fbOEERejectionReason1(
                        bEnable				:= TRUE,
                        bReset				:= ,
                        udiGlobalCounter	:= VIS.udiCounterGlobal, //Globalny licznik konfekcji [szt]
                        bAddReason			:= P13_BottleTransfer.fbBottleTransfer.eRunningState>1 AND VIS.nBottleTransferPlaceOption=2, // może dodać dodatkowy warunek?
                        bReason1			:= eRobotPackageState[1].bWeightTooLow 			AND eRobotPackageState[1].bBottlePresent,
                        sReason1Description	:= 'WZM',
                        bReason2			:= eRobotPackageState[1].bWeightTooHigh 		AND eRobotPackageState[1].bBottlePresent,
                        sReason2Description	:= 'WZD',
                        bReason3			:= NOT eRobotPackageState[1].bCapOK 			AND eRobotPackageState[1].bBottlePresent,
                        sReason3Description	:= 'BNPZ',
                        bReason4			:= NOT eRobotPackageState[1].bCapGripperScrewed AND eRobotPackageState[1].bBottlePresent,
                        sReason4Description	:= 'NZZSZ',
                        bReason5			:= NOT eRobotPackageState[1].bCapCorrectCapOn 	AND eRobotPackageState[1].bBottlePresent,
                        sReason5Description	:= 'BNZZ',
                        bReason6			:= eRobotPackageState[1].bCapCorrectNOK 		AND eRobotPackageState[1].bBottlePresent,
                        sReason6Description	:= 'NZZ',
                        bReason7			:=, 
                        sReason7Description	:= ,      
                        sRejectionReason	:= sOEERejectionReason1Temp,
                        );

fbOEERejectionReason2(
                        bEnable				:= TRUE,
                        bReset				:= ,
                        udiGlobalCounter	:= VIS.udiCounterGlobal, //Globalny licznik konfekcji [szt]
                        bAddReason			:= P13_BottleTransfer.fbBottleTransfer.eRunningState>1 AND VIS.nBottleTransferPlaceOption=2,
                        bReason1			:= eRobotPackageState[2].bWeightTooLow 			AND eRobotPackageState[2].bBottlePresent,
                        sReason1Description	:= 'WZM',
                        bReason2			:= eRobotPackageState[2].bWeightTooHigh 		AND eRobotPackageState[2].bBottlePresent,
                        sReason2Description	:= 'WZD',
                        bReason3			:= NOT eRobotPackageState[2].bCapOK 			AND eRobotPackageState[2].bBottlePresent,
                        sReason3Description	:= 'BNPZ',
                        bReason4			:= NOT eRobotPackageState[2].bCapGripperScrewed AND eRobotPackageState[2].bBottlePresent,
                        sReason4Description	:= 'NZZSZ',
                        bReason5			:= NOT eRobotPackageState[2].bCapCorrectCapOn 	AND eRobotPackageState[2].bBottlePresent,
                        sReason5Description	:= 'BNZZ',
                        bReason6			:= eRobotPackageState[2].bCapCorrectNOK 		AND eRobotPackageState[2].bBottlePresent,
                        sReason6Description	:= 'NZZ',
                        bReason7			:= , 
                        sReason7Description	:= ,      
                        sRejectionReason	:= sOEERejectionReason2Temp,
                        );
						
	rtfbOEERejectionReason2bDone(CLK:=fbOEERejectionReason2.bDone,Q=>);
	rtfbOEERejectionReason1bDone(CLK:=fbOEERejectionReason1.bDone,Q=>);
// dodałem na testy! 20.06	
	IF rtfbOEERejectionReason1bDone.Q AND  VIS.nBottleTransferPickOption=1 THEN
		VIS.sOEERejectionReason 			:=sOEERejectionReason1Temp;//	CONCAT(sOEERejectionReason1Temp,';');
		irtfbOEERejectionReason1bDoneCount	:=	irtfbOEERejectionReason1bDoneCount+1;
	END_IF
	
	
	IF rtfbOEERejectionReason2bDone.Q AND  VIS.nBottleTransferPickOption=2 THEN
		VIS.sOEERejectionReason 			:=	CONCAT(CONCAT(sOEERejectionReason1Temp,';'),sOEERejectionReason2Temp);
		irtfbOEERejectionReason2bDoneCount	:=	irtfbOEERejectionReason2bDoneCount+1;
	END_IF
	
    //Przeniesione dodawanie liczników, po to żeby dla wizualizacji i skryptów było łatwiej (kolejnosć odczytu)
    IF bAddGlobalCounter AND (fbOEERejectionReason2.bDone OR fbOEERejectionReason1.bDone )THEN
        VIS.uiCounterBadBottles                	:= VIS.uiCounterBadBottles		+ INT_TO_UINT(P00_PackML.nCounterFormsToLoad);//+ 1;// czy aby na pewno +1 ???
        VIS.udiCounterGlobalBadBottles        	:= VIS.udiCounterGlobalBadBottles	+ INT_TO_UDINT(P00_PackML.nCounterFormsToLoad);
        VIS.udiCounterGlobal                   	:= VIS.udiCounterGlobal			+ INT_TO_UDINT(P00_PackML.nCounterFormsToLoad);
        //VIS.udiCounterShiftBottles            	:= VIS.udiCounterShiftBottles	+ INT_TO_UDINT(P00_PackML.nCounterFormsToLoad);
        bAddGlobalCounter                    	:= FALSE;
    END_IF

    IF fbOEERejectionReason1.bAddReason THEN
       ifbOEERejectionReason1bAddReasonCount:=ifbOEERejectionReason1bAddReasonCount+1;
    END_IF
	
    IF fbOEERejectionReason2.bAddReason THEN
        ifbOEERejectionReason2bAddReasonCount:=ifbOEERejectionReason2bAddReasonCount+1;
     END_IF
END_ACTION

END_PROGRAM

// ---- POUs/FB/FB_OEECycleTimes.TcPOU
(*
Nazwa:			FB_OEECycleTimes
Opis:			czasy cyklów
Wersja:			v0.1
Data:			2021-11-09
Autor:			DP
Urzadzenia:		
Konfiguracja:	
Info: 
- dodano opcje przesuwu liniowego
*)
FUNCTION_BLOCK FB_OEECycleTimes
VAR_INPUT
	bEnable: BOOL;				//Zezwolenie na pracę
	bReset:BOOL;				//Stop awaryjny nieaktywny
	tStation1CT:TIME;			//Czas cyklu stacji nr 1
	bStation1En:BOOL;			//Zezwolenie pracy stacji nr 1
	sStation1Name:STRING;		//Nazwa stacji nr 1
	tStation2CT:TIME;			//Czas cyklu stacji nr 2
	bStation2En:BOOL;			//Zezwolenie pracy stacji nr 2
	sStation2Name:STRING;		//Nazwa stacji nr 2
	tStation3CT:TIME;			//Czas cyklu stacji nr 3
	bStation3En:BOOL;			//Zezwolenie pracy stacji nr 3
	sStation3Name:STRING;		//Nazwa stacji nr 3
	tStation4CT:TIME;			//Czas cyklu stacji nr 4
	bStation4En:BOOL;			//Zezwolenie pracy stacji nr 4
	sStation4Name:STRING;		//Nazwa stacji nr 4
	tStation5CT:TIME;			//Czas cyklu stacji nr 5
	bStation5En:BOOL;			//Zezwolenie pracy stacji nr 5
	sStation5Name:STRING;		//Nazwa stacji nr 5
	tStation6CT:TIME;			//Czas cyklu stacji nr 6
	bStation6En:BOOL;			//Zezwolenie pracy stacji nr 6
	sStation6Name:STRING;		//Nazwa stacji nr 6
	tStation7CT:TIME;			//Czas cyklu stacji nr 7
	bStation7En:BOOL;			//Zezwolenie pracy stacji nr 7
	sStation7Name:STRING;		//Nazwa stacji nr 7
	tStation8CT:TIME;			//Czas cyklu stacji nr 8
	bStation8En:BOOL;			//Zezwolenie pracy stacji nr 8
	sStation8Name:STRING;		//Nazwa stacji nr 8
	tStation9CT:TIME;			//Czas cyklu stacji nr 9
	bStation9En:BOOL;			//Zezwolenie pracy stacji nr 9
	sStation9Name:STRING;		//Nazwa stacji nr 9
	tStation10CT:TIME;			//Czas cyklu stacji nr 10
	bStation10En:BOOL;			//Zezwolenie pracy stacji nr 10
	sStation10Name:STRING;		//Nazwa stacji nr 10
	tStation11CT:TIME;			//Czas cyklu stacji nr 11
	bStation11En:BOOL;			//Zezwolenie pracy stacji nr 11
	sStation11Name:STRING;		//Nazwa stacji nr 11
	tStation12CT:TIME;			//Czas cyklu stacji nr 12
	bStation12En:BOOL;			//Zezwolenie pracy stacji nr 12
	sStation12Name:STRING;		//Nazwa stacji nr 12
	tStation13CT:TIME;			//Czas cyklu stacji nr 13
	bStation13En:BOOL;			//Zezwolenie pracy stacji nr 13
	sStation13Name:STRING;		//Nazwa stacji nr 13
	tStation14CT:TIME;			//Czas cyklu stacji nr 14
	bStation14En:BOOL;			//Zezwolenie pracy stacji nr 14
	sStation14Name:STRING;		//Nazwa stacji nr 14
	tStation15CT:TIME;			//Czas cyklu stacji nr 15
	bStation15En:BOOL;			//Zezwolenie pracy stacji nr 15	
	sStation15Name:STRING;		//Nazwa stacji nr 15
	tStation16CT:TIME;			//Czas cyklu stacji nr 16
	bStation16En:BOOL;			//Zezwolenie pracy stacji nr 16	
	sStation16Name:STRING;		//Nazwa stacji nr 16
	tStation17CT:TIME;			//Czas cyklu stacji nr 17
	bStation17En:BOOL;			//Zezwolenie pracy stacji nr 17	
	sStation17Name:STRING;		//Nazwa stacji nr 17
	tStation18CT:TIME;			//Czas cyklu stacji nr 18
	bStation18En:BOOL;			//Zezwolenie pracy stacji nr 18	
	sStation18Name:STRING;		//Nazwa stacji nr 18
	tStation19CT:TIME;			//Czas cyklu stacji nr 19
	bStation19En:BOOL;			//Zezwolenie pracy stacji nr 19	
	sStation19Name:STRING;		//Nazwa stacji nr 19
	tStation20CT:TIME;			//Czas cyklu stacji nr 20
	bStation20En:BOOL;			//Zezwolenie pracy stacji nr 20	
	sStation20Name:STRING;		//Nazwa stacji nr 20
	tStation21CT:TIME;			//Czas cyklu stacji nr 21
	bStation21En:BOOL;			//Zezwolenie pracy stacji nr 21	
	sStation21Name:STRING;		//Nazwa stacji nr 21	
	tStation22CT:TIME;			//Czas cyklu stacji nr 22
	bStation22En:BOOL;			//Zezwolenie pracy stacji nr 22	
	sStation22Name:STRING;		//Nazwa stacji nr 22	
	tStation23CT:TIME;			//Czas cyklu stacji nr 23
	bStation23En:BOOL;			//Zezwolenie pracy stacji nr 23	
	sStation23Name:STRING;		//Nazwa stacji nr 23	
	tStation24CT:TIME;			//Czas cyklu stacji nr 24
	bStation24En:BOOL;			//Zezwolenie pracy stacji nr 24	
	sStation24Name:STRING;		//Nazwa stacji nr 24	
	tStation25CT:TIME;			//Czas cyklu stacji nr 25
	bStation25En:BOOL;			//Zezwolenie pracy stacji nr 25	
	sStation25Name:STRING;		//Nazwa stacji nr 25	
	tStation26CT:TIME;			//Czas cyklu stacji nr 26
	bStation26En:BOOL;			//Zezwolenie pracy stacji nr 26	
	sStation26Name:STRING;		//Nazwa stacji nr 26	
	tStation27CT:TIME;			//Czas cyklu stacji nr 27
	bStation27En:BOOL;			//Zezwolenie pracy stacji nr 27	
	sStation27Name:STRING;		//Nazwa stacji nr 27	
	tStation28CT:TIME;			//Czas cyklu stacji nr 28
	bStation28En:BOOL;			//Zezwolenie pracy stacji nr 28	
	sStation28Name:STRING;		//Nazwa stacji nr 28	
	tStation29CT:TIME;			//Czas cyklu stacji nr 29
	bStation29En:BOOL;			//Zezwolenie pracy stacji nr 29	
	sStation29Name:STRING;		//Nazwa stacji nr 29	
	tStation30CT:TIME;			//Czas cyklu stacji nr 30
	bStation30En:BOOL;			//Zezwolenie pracy stacji nr 30	
	sStation30Name:STRING;		//Nazwa stacji nr 30	
	tStation31CT:TIME;			//Czas cyklu stacji nr 31
	bStation31En:BOOL;			//Zezwolenie pracy stacji nr 31	
	sStation31Name:STRING;		//Nazwa stacji nr 31	
	
END_VAR
VAR_OUTPUT
	AsCycleTimes					:ARRAY [0..63] OF STRING;		// Tabela czasów cykli 		[symbol_stacji;czas_w_ms]
END_VAR

VAR

END_VAR

ErrorHandling();
Cycle();
ManualMovements();
Statistics();

ACTION Cycle:


//Generowanie tablicy
IF tStation1CT < T#10S THEN	AsCycleTimes[1]:=	CONCAT(sStation1Name,	CONCAT(';',DINT_TO_STRING(TIME_TO_DINT(tStation1CT))));		ELSE tStation1CT := T#10S; END_IF;

IF tStation2CT < T#10S THEN	AsCycleTimes[2]:=	CONCAT(sStation2Name,	CONCAT(';',DINT_TO_STRING(TIME_TO_DINT(tStation2CT))));		ELSE tStation1CT := T#10S; END_IF;

IF tStation3CT < T#10S THEN	AsCycleTimes[3]:=	CONCAT(sStation3Name,	CONCAT(';',DINT_TO_STRING(TIME_TO_DINT(tStation3CT))));		ELSE tStation1CT := T#10S; END_IF;

IF tStation4CT < T#10S THEN	AsCycleTimes[4]:=	CONCAT(sStation4Name,	CONCAT(';',DINT_TO_STRING(TIME_TO_DINT(tStation4CT))));		ELSE tStation4CT := T#10S; END_IF;

IF tStation5CT < T#10S THEN	AsCycleTimes[5]:=	CONCAT(sStation5Name,	CONCAT(';',DINT_TO_STRING(TIME_TO_DINT(tStation5CT))));		ELSE tStation5CT := T#10S; END_IF;

IF tStation6CT < T#10S THEN	AsCycleTimes[6]:=	CONCAT(sStation6Name,	CONCAT(';',DINT_TO_STRING(TIME_TO_DINT(tStation6CT))));		ELSE tStation6CT := T#10S; END_IF;
	
IF tStation7CT < T#10S THEN AsCycleTimes[7]:=	CONCAT(sStation7Name,	CONCAT(';',DINT_TO_STRING(TIME_TO_DINT(tStation7CT))));		ELSE tStation7CT := T#10S; END_IF;
	
IF tStation8CT < T#10S THEN AsCycleTimes[8]:=	CONCAT(sStation8Name,	CONCAT(';',DINT_TO_STRING(TIME_TO_DINT(tStation8CT))));		ELSE tStation8CT := T#10S; END_IF;
	
IF tStation9CT < T#10S THEN AsCycleTimes[9]:=	CONCAT(sStation9Name,	CONCAT(';',DINT_TO_STRING(TIME_TO_DINT(tStation9CT))));		ELSE tStation9CT := T#10S; END_IF;
	
IF tStation10CT < T#10S THEN AsCycleTimes[10]:=	CONCAT(sStation10Name,	CONCAT(';',DINT_TO_STRING(TIME_TO_DINT(tStation10CT))));	ELSE tStation10CT := T#10S; END_IF;

IF tStation11CT < T#10S THEN AsCycleTimes[11]:=	CONCAT(sStation11Name,	CONCAT(';',DINT_TO_STRING(TIME_TO_DINT(tStation11CT))));	ELSE tStation11CT := T#10S; END_IF;

IF tStation12CT < T#10S THEN AsCycleTimes[12]:=	CONCAT(sStation12Name,	CONCAT(';',DINT_TO_STRING(TIME_TO_DINT(tStation12CT))));	ELSE tStation12CT := T#10S; END_IF;

IF tStation13CT < T#10S THEN AsCycleTimes[13]:=	CONCAT(sStation13Name,	CONCAT(';',DINT_TO_STRING(TIME_TO_DINT(tStation13CT))));	ELSE tStation13CT := T#10S; END_IF;

IF tStation14CT < T#10S THEN AsCycleTimes[14]:=	CONCAT(sStation14Name,	CONCAT(';',DINT_TO_STRING(TIME_TO_DINT(tStation14CT))));	ELSE tStation14CT := T#10S; END_IF;

IF tStation15CT < T#10S THEN AsCycleTimes[15]:=	CONCAT(sStation15Name,	CONCAT(';',DINT_TO_STRING(TIME_TO_DINT(tStation15CT))));	ELSE tStation15CT := T#10S; END_IF;

IF tStation16CT < T#10S THEN AsCycleTimes[16]:=	CONCAT(sStation16Name,	CONCAT(';',DINT_TO_STRING(TIME_TO_DINT(tStation16CT))));	ELSE tStation16CT := T#10S; END_IF;

IF tStation17CT < T#10S THEN AsCycleTimes[17]:=	CONCAT(sStation17Name,	CONCAT(';',DINT_TO_STRING(TIME_TO_DINT(tStation17CT))));	ELSE tStation17CT := T#10S; END_IF;

IF tStation18CT < T#10S THEN AsCycleTimes[18]:=	CONCAT(sStation18Name,	CONCAT(';',DINT_TO_STRING(TIME_TO_DINT(tStation18CT))));	ELSE tStation18CT := T#10S; END_IF;

IF tStation19CT < T#10S THEN AsCycleTimes[19]:=	CONCAT(sStation19Name,	CONCAT(';',DINT_TO_STRING(TIME_TO_DINT(tStation19CT))));	ELSE tStation19CT := T#10S; END_IF;

IF tStation20CT < T#10S THEN AsCycleTimes[20]:=	CONCAT(sStation20Name,	CONCAT(';',DINT_TO_STRING(TIME_TO_DINT(tStation20CT))));	ELSE tStation20CT := T#10S; END_IF;

IF tStation21CT < T#10S THEN AsCycleTimes[21]:=	CONCAT(sStation21Name,	CONCAT(';',DINT_TO_STRING(TIME_TO_DINT(tStation21CT))));	ELSE tStation21CT := T#10S; END_IF;

IF tStation22CT < T#10S THEN AsCycleTimes[22]:=	CONCAT(sStation22Name,	CONCAT(';',DINT_TO_STRING(TIME_TO_DINT(tStation22CT))));	ELSE tStation22CT := T#10S; END_IF;

IF tStation23CT < T#10S THEN AsCycleTimes[23]:=	CONCAT(sStation23Name,	CONCAT(';',DINT_TO_STRING(TIME_TO_DINT(tStation23CT))));	ELSE tStation23CT := T#10S; END_IF;
	
IF tStation24CT < T#10S THEN AsCycleTimes[24]:=	CONCAT(sStation24Name,	CONCAT(';',DINT_TO_STRING(TIME_TO_DINT(tStation24CT))));	ELSE tStation24CT := T#10S; END_IF;

IF tStation25CT < T#10S THEN AsCycleTimes[25]:=	CONCAT(sStation25Name,	CONCAT(';',DINT_TO_STRING(TIME_TO_DINT(tStation25CT))));	ELSE tStation25CT := T#10S; END_IF;

IF tStation26CT < T#10S THEN AsCycleTimes[26]:=	CONCAT(sStation26Name,	CONCAT(';',DINT_TO_STRING(TIME_TO_DINT(tStation26CT))));	ELSE tStation26CT := T#10S; END_IF;

IF tStation27CT < T#10S THEN AsCycleTimes[27]:=	CONCAT(sStation27Name,	CONCAT(';',DINT_TO_STRING(TIME_TO_DINT(tStation27CT))));	ELSE tStation27CT := T#10S; END_IF;

IF tStation28CT < T#10S THEN AsCycleTimes[28]:=	CONCAT(sStation28Name,	CONCAT(';',DINT_TO_STRING(TIME_TO_DINT(tStation28CT))));	ELSE tStation28CT := T#10S; END_IF;

IF tStation29CT < T#10S THEN AsCycleTimes[29]:=	CONCAT(sStation29Name,	CONCAT(';',DINT_TO_STRING(TIME_TO_DINT(tStation29CT))));	ELSE tStation29CT := T#10S; END_IF;

IF tStation30CT < T#10S THEN AsCycleTimes[30]:=	CONCAT(sStation30Name,	CONCAT(';',DINT_TO_STRING(TIME_TO_DINT(tStation30CT))));	ELSE tStation30CT := T#10S; END_IF;

IF tStation31CT < T#10S THEN AsCycleTimes[31]:=	CONCAT(sStation31Name,	CONCAT(';',DINT_TO_STRING(TIME_TO_DINT(tStation31CT))));	ELSE tStation31CT := T#10S; END_IF;
END_ACTION

ACTION ErrorHandling:

END_ACTION

ACTION ManualMovements:

END_ACTION

ACTION Statistics:

END_ACTION

END_FUNCTION_BLOCK

// ---- POUs/FB/FB_OEERejectionReason.TcPOU
(*
Nazwa:			FB_OEERejectionReasons
Opis:			Powód odrzuceń 
Wersja:			v0.1
Data:			2019-12-17
Autor:			DP
Urzadzenia:		
Konfiguracja:	
Info: 
- 
*)
FUNCTION_BLOCK FB_OEERejectionReason
VAR_INPUT
	bEnable: BOOL;				//Zezwolenie na pracę
	bReset:BOOL;				//Stop awaryjny nieaktywny
	udiGlobalCounter:UDINT;		//Globalny licznik
	bAddReason:BOOL;			//Dodaj pomiar
	bReason1:BOOL;
	sReason1Description:STRING;	//Nazwa stacji nr 1
	bReason2:BOOL;
	sReason2Description:STRING;	//Nazwa stacji nr 2
	bReason3:BOOL;
	sReason3Description:STRING;	//Nazwa stacji nr 3
	bReason4:BOOL;
	sReason4Description:STRING;	//Nazwa stacji nr 4
	bReason5:BOOL;
	sReason5Description:STRING;	//Nazwa stacji nr 5
	bReason6:BOOL;
	sReason6Description:STRING;	//Nazwa stacji nr 6
	bReason7:BOOL;
	sReason7Description:STRING;	//Nazwa stacji nr 7
	bReason8:BOOL;
	sReason8Description:STRING;	//Nazwa stacji nr 8
	bReason9:BOOL;
	sReason9Description:STRING;	//Nazwa stacji nr 9
	bReason10:BOOL;
	sReason10Description:STRING;	//Nazwa stacji nr 10
	bReason11:BOOL;
	sReason11Description:STRING;	//Nazwa stacji nr 11
	bReason12:BOOL;
	sReason12Description:STRING;	//Nazwa stacji nr 12
	bReason13:BOOL;
	sReason13Description:STRING;	//Nazwa stacji nr 13
	bReason14:BOOL;
	sReason14Description:STRING;	//Nazwa stacji nr 14
END_VAR

VAR_IN_OUT
	sRejectionReason			:STRING;		// Powodu odrzuceń	[symbol_odrzucenia] narazie tylko w tabeli 1
END_VAR
VAR_OUTPUT
	bDone						:BOOL;		// Powodu odrzuceń	[symbol_odrzucenia] narazie tylko w tabeli 1
END_VAR

VAR
	rtAddReason: R_TRIG;
	tonResetDone: TON;
END_VAR

ErrorHandling();
Cycle();
ManualMovements();
Statistics();

ACTION Cycle:
tonResetDone(IN:=bDone,PT:=T#300MS);
rtAddReason(CLK:=bAddReason,Q=>);
IF rtAddReason.Q THEN
	IF bReason1 THEN
		sRejectionReason:= sReason1Description;
	ELSIF bReason2 THEN		                
		sRejectionReason:= sReason2Description;
	ELSIF bReason3 THEN		                
		sRejectionReason:= sReason3Description;
	ELSIF bReason4 THEN		                
		sRejectionReason:= sReason4Description;
	ELSIF bReason5 THEN		                
		sRejectionReason:= sReason5Description;
	ELSIF bReason6 THEN		                
		sRejectionReason:= sReason6Description;
	ELSIF bReason7 THEN		                
		sRejectionReason:= sReason7Description;
	ELSIF bReason8 THEN		                
		sRejectionReason:= sReason8Description;
	ELSIF bReason9 THEN		                
		sRejectionReason:= sReason9Description;
	ELSIF bReason10 THEN		                
		sRejectionReason:= sReason10Description;
	ELSIF bReason11 THEN		                
		sRejectionReason:= sReason11Description;
	ELSIF bReason12 THEN		                
		sRejectionReason:= sReason12Description;
	ELSIF bReason13 THEN		                
		sRejectionReason:= sReason13Description;
	ELSIF bReason14 THEN		                
		sRejectionReason:= sReason14Description;

	END_IF
	bDone:= TRUE;
END_IF
IF tonResetDone.Q THEN
	bDone:= FALSE;
END_IF
END_ACTION

ACTION ErrorHandling:

END_ACTION

ACTION ManualMovements:

END_ACTION

ACTION Statistics:

END_ACTION

END_FUNCTION_BLOCK

// ---- POUs/P00_Recipes.TcPOU
PROGRAM P00_Recipes
(*
Nazwa:			P_Recipes
Wersja:			v0.1 			
Autor:			TW,DP
Urzadzenia:		HMI, 
Konfiguracja:	
Info:
- 50 receptur
- sortowanie
- odczytwanie, zapisywanie jako nowa, aktualizacja, usuwanie, wybór
- receptura 1 jako ustawienia fabryczne
Uwagi:
- na końcu aktualizować nastawy pierwszej receptury
Zmiany:
2018-05-07 DP Dodano na stałe wpisywanie danych do pierwszej receptury
*)
VAR
	i: INT;
	h: INT;
	bTestDwuFaz: BOOL;
	iLidSealerTempHisteresis: INT;
	bTestTransporter: BOOL;
	fbiPackageNozzleDiameter:FB_Skalowanie;
	rPackageNozzleDiameterFactor:REAL;	
	rPackageMassTypeFactor:REAL;	
END_VAR

//wybór programu
IF VIS.bChooseRecipe THEN
	IF VIS.bDialogBoxAck THEN
		VIS.bChooseRecipe := FALSE;
		VIS.bDialogBoxAck:=FALSE;
		bRecipeAfterPowerStateChosen := TRUE; //Wybrano pierwszą recepturę po ruchomieniu
	ELSIF VIS.bDialogBoxCancelAck THEN
		VIS.bDialogBoxAck:=FALSE;
		VIS.bChooseRecipe := FALSE;
		VIS.bDialogBoxCancelAck:=FALSE;
	END_IF
END_IF

(*Automatyczne ustawianie danych receptur*)
aAutoSetRecipeParameters();

(*dane receptur*)
aShowToAll();
aTwoSpeeds();
aLimits();	
//Receptura fabryczna
//Na stałe bez możliwości zmiany
//Zawsze można zapisać jako inną i tam zmieniać parametry
VIS.bChooseRecipe;
VIS.bDialogBoxAck;
IF NOT bFirstPositioningDone  THEN						//do skomentowania Vasyl
	aFactoryRecipes();
END_IF
IF bHomingCanceled AND NOT bFirstPositioningDone THEN
	bFirstPositioningDone	:= TRUE;
END_IF

ACTION aAutoSetRecipeParameters:

(****************** AUTO DOSTRAJANIE CZASÓW TRANSPORTERÓW*********)
	//Czas przy najwolnejszej prędkości transportera 15Hz
	//15Hz 300 2000ms
	//25Hz 500 1300ms
	//35Hz 700 1000ms
	//45Hz 900 700ms
	//56Hz 1100 600ms
	//67Hz 1300 500ms
	// Wyznaczona funkcja potęgowa
	IF GVL.nFormTransportersDispencerVelocitySV > 0 AND GVL.nFormTransportersDispencerVelocitySV <1000 THEN
		
		VIS.nGateBeforeDispencersTimeFormInsertingShow := 500;
		(*nExitWheelFormsTime := LREAL_TO_UINT(
										850601 * EXPT(nFormTransportersVelocitySV,-0.94)
											);*)										
		{warning 'Czasy otwarcia narazie na stałe-sprawdzić dla szybkiej i najwolniejszej prędkości transportera}			
	ELSE
		VIS.nGateBeforeDispencersTimeFormInsertingShow := 300;
		(*nExitWheelFormsTime := LREAL_TO_UINT(
										850601 * EXPT(nFormTransportersVelocitySV,-0.94)
											);*)										
			;
	END_IF
	
	IF 		GVL.nFormTransportersDispencerVelocitySV 	>	1100	THEN			
				VIS.nGateRobotTimeFormInsertingShow		:= 300;	//bylo 300	
	ELSIF 		GVL.nFormTransportersDispencerVelocitySV 	>	1000	THEN			
				VIS.nGateRobotTimeFormInsertingShow		:= 300;		
	ELSIF	GVL.nFormTransportersDispencerVelocitySV 	>	900		THEN
				VIS.nGateRobotTimeFormInsertingShow		:= 400;		
	ELSIF	GVL.nFormTransportersDispencerVelocitySV 	>	800		THEN
				VIS.nGateRobotTimeFormInsertingShow		:= 450;		
	ELSIF	GVL.nFormTransportersDispencerVelocitySV 	>	700		THEN
				VIS.nGateRobotTimeFormInsertingShow		:= 600;	
	ELSIF	GVL.nFormTransportersDispencerVelocitySV 	>	600		THEN
				VIS.nGateRobotTimeFormInsertingShow		:= 800;	
	ELSIF	GVL.nFormTransportersDispencerVelocitySV 	>	500		THEN
				VIS.nGateRobotTimeFormInsertingShow		:= 900;	
	ELSE
			VIS.nGateRobotTimeFormInsertingShow		:= 1000;	
	END_IF	
	
	
	
	//Parametry opakowania  [Ekran obliczania parametrów]
    //[[[[[[[[[[[[[[[[[[[[[[[[[[[[[[[[[[[[[[[[[[[[[[[[[[[
 	VIS.iPackagePuckInsertHeightShow;// Wysokość wkładki w formatce (0-100mm)  (samej wkładki) (Do pozycji odkładania robota)              
  	VIS.iPackageMassTypeShow		;// Typ masy 	(0-Woda, 1-Olej, 2-Mydło, 3-Krem itd.)
	VIS.iPackageCapTypeShow			;// Typ nasadki (0-Fliptop, 1-Pompka/Atomizer, 2-Kulka, 3-Airless, 4-, 5- Deko, 6-Nakrętka_słoika
	VIS.iPackageCapDiameterShow		;// Średnica nasadki (5-100mm),
	VIS.iPackageHeightShow			;// Wysokość butelki razem z formatką (50-300mm),	
	VIS.iPackageCappedHeightShow	;// Wysokość butelki razem z dokręconą nakrętką i formatką (50-350mm),		
	VIS.iPackageNozzleDiameterShow	;// Srednica zewnetrzna wylewki (5-30mm),	
	VIS.lrDispencer1DoseVolumeShow  ;// Ilość dozy (10-560ml)
 	VIS.lrCupWeightShow	 			;// Waga opakowania (0-500g)
 	VIS.bRecipeCalculate;			 // Oblicz
	 //[[[[[[[[[[[[[[[[[[[[[[[[[[[[[[[[[[[[[[[[[[[[[[[[[[[
	 
	// Limity
	 IF VIS.iPackageHeightShow = 0 			THEN VIS.iPackageHeightShow := 150;	 			END_IF
	 IF VIS.iPackageCappedHeightShow = 0 	THEN VIS.iPackageCappedHeightShow := 160;		END_IF	 
	 IF VIS.iPackageNozzleDiameterShow = 0 	THEN VIS.iPackageNozzleDiameterShow := 16;		END_IF	 
	
	// Skalowanie - Prędkość Dozowania <-> Średnica wylewki
	 rPackageNozzleDiameterFactor := 						1.4285 * EXPT(VIS.iPackageNozzleDiameterShow,1.5615);	
	// Skalowanie - Typ masy 	(0-Woda, 1-Olej, 2-Mydło, 3-Krem itd.)
	IF   	VIS.iPackageMassTypeShow	= 0 THEN	rPackageMassTypeFactor := 1.0;
	ELSIF	VIS.iPackageMassTypeShow	= 1 THEN	rPackageMassTypeFactor := 0.8;
	ELSIF	VIS.iPackageMassTypeShow	= 2 THEN	rPackageMassTypeFactor := 1.3;
	ELSIF	VIS.iPackageMassTypeShow	= 3 THEN	rPackageMassTypeFactor := 1.5;		END_IF
	// Prędkość dozowania
	rPackageNozzleDiameterFactor; (**) rPackageMassTypeFactor;
	
	// Oblicz
	IF VIS.bRecipeCalculate THEN
					
        //Podawanie butelekButelki                                  
		VIS.lrPucksInserterHammerHeightSVShow				:=	VIS.iPackageHeightShow+1;                                            				                                                                                                                           																		
       
		//Dozownik	                             	                                                                                     												
		VIS.lrDispencersLifterReadyPositionShow				:=	VIS.iPackageHeightShow + 60;                                                                                             
		VIS.lrDispencer1LifterStartDosePositionShow			:=	VIS.iPackagePuckInsertHeightShow + 29 + 25;                                           
		VIS.lrDispencer1LifterStopDosePositionShow			:=	VIS.iPackageHeightShow - 10;                                                                                  
		VIS.lrDispencersCatchHeightSVShow					:=	VIS.iPackageHeightShow - 5;                                                  
       	IF  VIS.iPackageMassTypeShow = 0 THEN // (0-Woda, 1-Olej, 2-Mydło, 3-Krem itd.)                               
			VIS.lrDispencer1Phase1VolumeShow				:=	FLOOR(VIS.lrDispencer1DoseVolumeShow*0.2);                                          
			VIS.lrDispencer1Phase2VolumeShow				:=	0;
			VIS.lrDispencer1Phase1VelocityShow				:=	rPackageNozzleDiameterFactor * rPackageMassTypeFactor * 0.7;
			VIS.lrDispencer1Phase2VelocityShow				:=	rPackageNozzleDiameterFactor * rPackageMassTypeFactor;
			VIS.lrDispencer1Phase3VelocityShow				:=	rPackageNozzleDiameterFactor * rPackageMassTypeFactor * 0.7;
			VIS.lrDispencer1SuckVelocityShow				:=	200;
			VIS.lrDispencer1Phase1AccelerationShow			:=	300;
			VIS.lrDispencer1Phase2AccelerationShow			:=	400;
			VIS.lrDispencer1Phase3AccelerationShow			:=	50;
			VIS.lrDispencer1SuckAccelerationShow			:=	3000;
			VIS.lrDispencer1Phase1DecelerationShow			:=	150;
			VIS.lrDispencer1Phase2DecelerationShow			:=	1000;
			VIS.lrDispencer1Phase3DecelerationShow			:=	50;
			VIS.udiDispencer1DosingDoneDelayTimeShow		:=	100;
			VIS.lrDispencer1SuckValveOpenVolumeShow			:=	0;
			VIS.lrDispencer1SuckValveOpenTimeDelayShow		:=	0;
			VIS.lrDispencer1SuckValveCloseVolumeShow		:=	0;
			VIS.lrDispencer1SuckValveCloseTimeDelayShow		:=	0;
			VIS.lrDispencer1DoseValveOpenVolumeShow			:=	0;
			VIS.lrDispencer1DoseValveOpenTimeAccShow		:=	100;
			VIS.lrDispencer1DoseValveCloseVolumeShow		:=	0;
			VIS.lrDispencer1DoseValveCloseTimeDecShow		:=	0;
			VIS.lrDispencer1DoseSuckingVolumeShow			:=	0;
			VIS.lrDispencer1DoseSuckingTimeDelayShow		:=	0;
			VIS.bDispencer1DoseSuckingShow					:=	FALSE;
			VIS.bDispencer2LiftSynchroPh1Show				:=	FALSE;
			VIS.bDispencer2LiftSynchroPh2Show				:=	TRUE;
			VIS.bDispencer2LiftSynchroPh3Show				:=	TRUE;	
		ELSIF VIS.iPackageMassTypeShow = 1 THEN // (0-Woda, 1-Olej, 2-Mydło, 3-Krem itd.)   
			VIS.lrDispencer1Phase1VolumeShow				:=	FLOOR(VIS.lrDispencer1DoseVolumeShow*0.2);                                          
			VIS.lrDispencer1Phase2VolumeShow				:=	FLOOR(VIS.lrDispencer1DoseVolumeShow*0.2); 
			VIS.lrDispencer1Phase1VelocityShow				:=	rPackageNozzleDiameterFactor * rPackageMassTypeFactor * 0.7;
			VIS.lrDispencer1Phase2VelocityShow				:=	rPackageNozzleDiameterFactor * rPackageMassTypeFactor;
			VIS.lrDispencer1Phase3VelocityShow				:=	rPackageNozzleDiameterFactor * rPackageMassTypeFactor * 0.7;
			VIS.lrDispencer1SuckVelocityShow				:=	100;
			VIS.lrDispencer1Phase1AccelerationShow			:=	40;
			VIS.lrDispencer1Phase2AccelerationShow			:=	50;
			VIS.lrDispencer1Phase3AccelerationShow			:=	40;
			VIS.lrDispencer1SuckAccelerationShow			:=	500;
			VIS.lrDispencer1Phase1DecelerationShow			:=	80;
			VIS.lrDispencer1Phase2DecelerationShow			:=	100;
			VIS.lrDispencer1Phase3DecelerationShow			:=	80;
			VIS.udiDispencer1DosingDoneDelayTimeShow		:=	200;
			VIS.lrDispencer1SuckValveOpenVolumeShow			:=	0;
			VIS.lrDispencer1SuckValveOpenTimeDelayShow		:=	0;
			VIS.lrDispencer1SuckValveCloseVolumeShow		:=	0;
			VIS.lrDispencer1SuckValveCloseTimeDelayShow		:=	0;
			VIS.lrDispencer1DoseValveOpenVolumeShow			:=	0;
			VIS.lrDispencer1DoseValveOpenTimeAccShow		:=	200;
			VIS.lrDispencer1DoseValveCloseVolumeShow		:=	0;
			VIS.lrDispencer1DoseValveCloseTimeDecShow		:=	0;
			VIS.lrDispencer1DoseSuckingVolumeShow			:=	0;
			VIS.lrDispencer1DoseSuckingTimeDelayShow		:=	0;
			VIS.bDispencer1DoseSuckingShow					:=	FALSE;
			VIS.bDispencer2LiftSynchroPh1Show				:=	TRUE;
			VIS.bDispencer2LiftSynchroPh2Show				:=	TRUE;
			VIS.bDispencer2LiftSynchroPh3Show				:=	TRUE;	
		ELSIF VIS.iPackageMassTypeShow = 2 THEN // (0-Woda, 1-Olej, 2-Mydło, 3-Krem itd.)   
			VIS.lrDispencer1Phase1VolumeShow				:=	FLOOR(VIS.lrDispencer1DoseVolumeShow*0.2);                                          
			VIS.lrDispencer1Phase2VolumeShow				:=	0;
			VIS.lrDispencer1Phase1VelocityShow				:=	rPackageNozzleDiameterFactor * rPackageMassTypeFactor * 0.7;
			VIS.lrDispencer1Phase2VelocityShow				:=	rPackageNozzleDiameterFactor * rPackageMassTypeFactor;      
			VIS.lrDispencer1Phase3VelocityShow				:=	rPackageNozzleDiameterFactor * rPackageMassTypeFactor * 0.7;
			VIS.lrDispencer1SuckVelocityShow				:=	200;
			VIS.lrDispencer1Phase1AccelerationShow			:=	300;
			VIS.lrDispencer1Phase2AccelerationShow			:=	400;
			VIS.lrDispencer1Phase3AccelerationShow			:=	50;
			VIS.lrDispencer1SuckAccelerationShow			:=	3000;
			VIS.lrDispencer1Phase1DecelerationShow			:=	150;
			VIS.lrDispencer1Phase2DecelerationShow			:=	1000;
			VIS.lrDispencer1Phase3DecelerationShow			:=	50;
			VIS.udiDispencer1DosingDoneDelayTimeShow		:=	200;
			VIS.lrDispencer1SuckValveOpenVolumeShow			:=	0;
			VIS.lrDispencer1SuckValveOpenTimeDelayShow		:=	0;
			VIS.lrDispencer1SuckValveCloseVolumeShow		:=	0;
			VIS.lrDispencer1SuckValveCloseTimeDelayShow		:=	0;
			VIS.lrDispencer1DoseValveOpenVolumeShow			:=	0;
			VIS.lrDispencer1DoseValveOpenTimeAccShow		:=	200;
			VIS.lrDispencer1DoseValveCloseVolumeShow		:=	0;
			VIS.lrDispencer1DoseValveCloseTimeDecShow		:=	0;
			VIS.lrDispencer1DoseSuckingVolumeShow			:=	0;
			VIS.lrDispencer1DoseSuckingTimeDelayShow		:=	0;
			VIS.bDispencer1DoseSuckingShow					:=	FALSE;
			VIS.bDispencer2LiftSynchroPh1Show				:=	FALSE;
			VIS.bDispencer2LiftSynchroPh2Show				:=	TRUE;
			VIS.bDispencer2LiftSynchroPh3Show				:=	TRUE;	
		ELSIF VIS.iPackageMassTypeShow = 3 THEN // (0-Woda, 1-Olej, 2-Mydło, 3-Krem itd.)   
			VIS.lrDispencer1Phase1VolumeShow				:=	FLOOR(VIS.lrDispencer1DoseVolumeShow*0.2);                                          
			VIS.lrDispencer1Phase2VolumeShow				:=	0;
			VIS.lrDispencer1Phase1VelocityShow				:=	rPackageNozzleDiameterFactor * rPackageMassTypeFactor * 0.7;
			VIS.lrDispencer1Phase2VelocityShow				:=	rPackageNozzleDiameterFactor * rPackageMassTypeFactor;      
			VIS.lrDispencer1Phase3VelocityShow				:=	rPackageNozzleDiameterFactor * rPackageMassTypeFactor * 0.7;
			VIS.lrDispencer1SuckVelocityShow				:=	200;
			VIS.lrDispencer1Phase1AccelerationShow			:=	300;
			VIS.lrDispencer1Phase2AccelerationShow			:=	400;
			VIS.lrDispencer1Phase3AccelerationShow			:=	50;
			VIS.lrDispencer1SuckAccelerationShow			:=	3000;
			VIS.lrDispencer1Phase1DecelerationShow			:=	150;
			VIS.lrDispencer1Phase2DecelerationShow			:=	1000;
			VIS.lrDispencer1Phase3DecelerationShow			:=	50;
			VIS.udiDispencer1DosingDoneDelayTimeShow		:=	200;
			VIS.lrDispencer1SuckValveOpenVolumeShow			:=	0;
			VIS.lrDispencer1SuckValveOpenTimeDelayShow		:=	0;
			VIS.lrDispencer1SuckValveCloseVolumeShow		:=	0;
			VIS.lrDispencer1SuckValveCloseTimeDelayShow		:=	0;
			VIS.lrDispencer1DoseValveOpenVolumeShow			:=	0;
			VIS.lrDispencer1DoseValveOpenTimeAccShow		:=	200;
			VIS.lrDispencer1DoseValveCloseVolumeShow		:=	0;
			VIS.lrDispencer1DoseValveCloseTimeDecShow		:=	0;
			VIS.lrDispencer1DoseSuckingVolumeShow			:=	0;
			VIS.lrDispencer1DoseSuckingTimeDelayShow		:=	0;
			VIS.bDispencer1DoseSuckingShow					:=	FALSE;
			VIS.bDispencer2LiftSynchroPh1Show				:=	FALSE;
			VIS.bDispencer2LiftSynchroPh2Show				:=	TRUE;
			VIS.bDispencer2LiftSynchroPh3Show				:=	TRUE;	
		END_IF

		//Chwytak butelek
		VIS.lrDispencersCatch1ClosedValueShow				:= VIS.iPackageCapDiameterShow-1;
		VIS.lrDispencersCatch1OpenValueShow					:= 58;
		VIS.lrDispencersCatch2ClosedValueShow				:= VIS.iPackageCapDiameterShow+2;
		VIS.lrDispencersCatch2OpenValueShow					:= 60.2;
		VIS.lrDispencersCatch3ClosedValueShow				:= VIS.iPackageCapDiameterShow+2;
		VIS.lrDispencersCatch3OpenValueShow					:= 60.1;
		VIS.lrDispencersCatch4ClosedValueShow				:= VIS.iPackageCapDiameterShow-1;
		VIS.lrDispencersCatch4OpenValueShow					:= 55.6;
		VIS.lrDispencersCatchToleranceShow					:= 15;
	
		//Waga
		VIS.lrWeightMassSVShow								:= VIS.lrDispencer1DoseVolumeShow;
		VIS.lrWeightUpperToleranceShow						:= FLOOR(VIS.lrDispencer1DoseVolumeShow * 0.02);	
		VIS.lrWeightLowerToleranceShow						:= FLOOR(VIS.lrDispencer1DoseVolumeShow * 0.03);	
		                                                                                                                                                                       		                                                                                        
		//Podajnik platynek                                                                     	                                
		VIS.lrLidFeederHeightPosSVShow						:=	VIS.iPackageHeightShow + 5;  				                                
						                            	                            
		//Sprawdzanie platynek				
		VIS.lrLidPuttedCheckHeightSVShow					:=	VIS.iPackageHeightShow + 5;  	 			
					
		//Zgrzewanie				
		VIS.lrLidSealerHeightPosSVShow						:=	VIS.iPackageHeightShow + 5;  								
		
		//ROPP-Podajnik                                    		
		VIS_ROPP.lrROPPFeederHeightPosSVShow				:=	VIS.iPackageHeightShow + 5;                                                      
		//ROPP-Zakrecanie                    		
		VIS_ROPP.lrROPPCappingHeightPosSVShow				:=	VIS.iPackageHeightShow + 5;  
		
		//Podajnik nakrętek
		VIS.lrCapFeederHeightPosSVShow						:=	VIS.iPackageHeightShow + 12;  		

		//Test nasadki	// Typ nasadki (0-Fliptop, 1-Pompka/Atomizer, 2-Kulka, 3-Airless, 4-, 5- Deko, 6-Nakrętka_słoika
		IF 		VIS.iPackageCapTypeShow	= 0 THEN 			VIS.lrCapPuttedCheckHeightPosSVShow	:=	VIS.iPackageHeightShow ;  
		ELSIF 	VIS.iPackageCapTypeShow	= 1 THEN 			VIS.lrCapPuttedCheckHeightPosSVShow	:=	VIS.iPackageHeightShow ;  	
		ELSIF 	VIS.iPackageCapTypeShow	= 2 THEN 			VIS.lrCapPuttedCheckHeightPosSVShow	:=	VIS.iPackageHeightShow ;   
		ELSIF 	VIS.iPackageCapTypeShow	= 3 THEN 			VIS.lrCapPuttedCheckHeightPosSVShow	:=	VIS.iPackageHeightShow ;  
		ELSIF 	VIS.iPackageCapTypeShow	= 4 THEN 			VIS.lrCapPuttedCheckHeightPosSVShow	:=	VIS.iPackageHeightShow ;  
		ELSIF 	VIS.iPackageCapTypeShow	= 5 THEN 			VIS.lrCapPuttedCheckHeightPosSVShow	:=	VIS.iPackageHeightShow ;  
		ELSIF 	VIS.iPackageCapTypeShow	= 6 THEN 			VIS.lrCapPuttedCheckHeightPosSVShow	:=	VIS.iPackageHeightShow ;  
		END_IF	

		//Zakręcarka
		IF 	VIS.iPackageCapTypeShow	= 0 THEN // Typ nasadki (0-Fliptop, 1-Pompka/Atomizer, 2-Kulka, 3-Airless, 4-, 5- Deko, 6-Nakrętka_słoika
			VIS.lrGripperScrewingTightTorqueShow				:=	0.5;
			VIS.lrGripperScrewing2TightTorqueShow				:=	0.5;
			VIS.iGripperScrewer1ToolShow						:=	0; //0-Dwu,1-Trój,2-Kształtowa/DoKulek,3-Wbijająca,4-Zasysająca
			VIS.lrGripperScrewer1VelocityShow					:=	90;
			VIS.nGripperScrewer1TightTimeShow					:=	300;
			VIS.lrGripperScrewerReadyPositionShow				:=	VIS.iPackageHeightShow + 14;	
			VIS.lrGripperScrewerPushingCapPositionShow			:=	VIS.iPackageHeightShow + 14;	
			VIS.lrGripperScrewerScrewingCapPositionShow			:=	VIS.iPackageHeightShow + 14;
			VIS.lrGripperScrewerFindScrewPositionShow			:=	VIS.iPackageHeightShow + 14;	
			VIS.lrGripperScrewerPressureShow					:=	15;
			VIS.lrGripperScrewerCatchPressureShow				:=	7;
			VIS.lrGripperScrewerPressureExhaustLevelShow		:=	100.0;
			VIS.lrGripperScrewerCatchPressureExhaustLevelShow	:=	100.0;
			VIS.lrGripperScrewerTurnoversToFullScrewedShow		:=	1;
			VIS.lrGripperScrewerThreadPitchShow					:=	3;			
			VIS.lrGripperScrewerThreadTimesShow					:=	1.0;		
			VIS.nGripperScrewerCatchHeightSVShow				:=	VIS_M.iPuckHeight + 10;
			VIS.bGripperScrewer1FindScrewShow					:=	FALSE;
			VIS.bGripperScrewer1Option4Show						:=	FALSE;
			VIS.lrGripperScrewer1FindingScrewDegreeShow			:=	260;
			VIS.bGripperScrewer1Option1Show						:=	FALSE;
			VIS.bGripperScrewer1Option2Show						:=	FALSE;
			VIS.bGripperScrewer1Option3Show						:=	TRUE;
			VIS.bGripperScrewer1Option5Show						:=	FALSE;
			VIS.bGripperScrewer1Option6Show						:=	TRUE;
			VIS.bGripperScrewer1Option7Show						:=	TRUE;
		ELSIF VIS.iPackageCapTypeShow	= 1 THEN // Typ nasadki (0-Fliptop, 1-Pompka/Atomizer, 2-Kulka, 3-Airless, 4-, 5- Deko, 6-Nakrętka_słoika
			VIS.lrGripperScrewingTightTorqueShow				:=	0.5;
			VIS.lrGripperScrewing2TightTorqueShow				:=	0.5;
			VIS.iGripperScrewer1ToolShow						:=	0;//0-Dwu,1-Trój,2-Kształtowa/DoKulek,3-Wbijająca,4-Zasysająca
			VIS.lrGripperScrewer1VelocityShow					:=	90;
			VIS.nGripperScrewer1TightTimeShow					:=	300;
			VIS.lrGripperScrewerReadyPositionShow				:=	VIS.iPackageHeightShow + 25;	
			VIS.lrGripperScrewerPushingCapPositionShow			:=	VIS.iPackageHeightShow + 14;	
			VIS.lrGripperScrewerScrewingCapPositionShow			:=	VIS.iPackageHeightShow + 14;	
			VIS.lrGripperScrewerFindScrewPositionShow			:=	VIS.iPackageHeightShow + 14;
			VIS.lrGripperScrewerPressureShow					:=	30;
			VIS.lrGripperScrewerCatchPressureShow				:=	20;
			VIS.lrGripperScrewerPressureExhaustLevelShow		:=	100.0;
			VIS.lrGripperScrewerCatchPressureExhaustLevelShow	:=	100.0;
			VIS.lrGripperScrewerTurnoversToFullScrewedShow		:=	1;
			VIS.lrGripperScrewerThreadPitchShow					:=	3;			
			VIS.lrGripperScrewerThreadTimesShow					:=	1.0;		
			VIS.nGripperScrewerCatchHeightSVShow				:=	110;
			VIS.bGripperScrewer1FindScrewShow					:=	FALSE;
			VIS.bGripperScrewer1Option4Show						:=	FALSE;
			VIS.lrGripperScrewer1FindingScrewDegreeShow			:=	260;
			VIS.bGripperScrewer1Option1Show						:=	FALSE;
			VIS.bGripperScrewer1Option2Show						:=	FALSE;
			VIS.bGripperScrewer1Option3Show						:=	TRUE;
			VIS.bGripperScrewer1Option5Show						:=	FALSE;
			VIS.bGripperScrewer1Option6Show						:=	TRUE;
			VIS.bGripperScrewer1Option7Show						:=	TRUE;
		ELSIF VIS.iPackageCapTypeShow	= 2 THEN // Typ nasadki (0-Fliptop, 1-Pompka/Atomizer, 2-Kulka, 3-Airless, 4-, 5- Deko, 6-Nakrętka_słoika
			VIS.lrGripperScrewingTightTorqueShow				:=	0.5;
			VIS.lrGripperScrewing2TightTorqueShow				:=	0.5;
			VIS.iGripperScrewer1ToolShow						:=	2;//0-Dwu,1-Trój,2-Kształtowa/DoKulek,3-Wbijająca,4-Zasysająca
			VIS.lrGripperScrewer1VelocityShow					:=	90;
			VIS.nGripperScrewer1TightTimeShow					:=	300;
			VIS.lrGripperScrewerReadyPositionShow				:=	VIS.iPackageHeightShow + 30;	
			VIS.lrGripperScrewerPushingCapPositionShow			:=	VIS.iPackageHeightShow - 10;	
			VIS.lrGripperScrewerScrewingCapPositionShow			:=	VIS.iPackageHeightShow - 10;
			VIS.lrGripperScrewerFindScrewPositionShow			:=	VIS.iPackageHeightShow - 10;	
			VIS.lrGripperScrewerPressureShow					:=	30;
			VIS.lrGripperScrewerCatchPressureShow				:=	20;
			VIS.lrGripperScrewerPressureExhaustLevelShow		:=	100.0;
			VIS.lrGripperScrewerCatchPressureExhaustLevelShow	:=	100.0;
			VIS.lrGripperScrewerTurnoversToFullScrewedShow		:=	1;
			VIS.lrGripperScrewerThreadPitchShow					:=	3;			
			VIS.lrGripperScrewerThreadTimesShow					:=	1.0;		
			VIS.nGripperScrewerCatchHeightSVShow				:=	110;
			VIS.bGripperScrewer1FindScrewShow					:=	FALSE;
			VIS.bGripperScrewer1Option4Show						:=	FALSE;
			VIS.lrGripperScrewer1FindingScrewDegreeShow			:=	260;
			VIS.bGripperScrewer1Option1Show						:=	FALSE;
			VIS.bGripperScrewer1Option2Show						:=	FALSE;
			VIS.bGripperScrewer1Option3Show						:=	TRUE;
			VIS.bGripperScrewer1Option5Show						:=	FALSE;
			VIS.bGripperScrewer1Option6Show						:=	TRUE;
			VIS.bGripperScrewer1Option7Show						:=	TRUE;
		ELSIF VIS.iPackageCapTypeShow	= 3 THEN // Typ nasadki (0-Fliptop, 1-Pompka/Atomizer, 2-Kulka, 3-Airless, 4-, 5- Deko, 6-Nakrętka_słoika
			VIS.lrGripperScrewingTightTorqueShow				:=	0.5;
			VIS.lrGripperScrewing2TightTorqueShow				:=	0.5;
			VIS.iGripperScrewer1ToolShow						:=	3;//0-Dwu,1-Trój,2-Kształtowa/DoKulek,3-Wbijająca,4-Zasysająca
			VIS.lrGripperScrewer1VelocityShow					:=	90;
			VIS.nGripperScrewer1TightTimeShow					:=	300;
			VIS.lrGripperScrewerReadyPositionShow				:=	VIS.iPackageHeightShow + 60;	
			VIS.lrGripperScrewerPushingCapPositionShow			:=	VIS.iPackageHeightShow + 14;	
			VIS.lrGripperScrewerScrewingCapPositionShow			:=	VIS.iPackageHeightShow + 14;	
			VIS.lrGripperScrewerFindScrewPositionShow			:=	VIS.iPackageHeightShow + 14;
			VIS.lrGripperScrewerPressureShow					:=	30;
			VIS.lrGripperScrewerCatchPressureShow				:=	20;
			VIS.lrGripperScrewerPressureExhaustLevelShow		:=	100.0;
			VIS.lrGripperScrewerCatchPressureExhaustLevelShow	:=	100.0;
			VIS.lrGripperScrewerTurnoversToFullScrewedShow		:=	1;
			VIS.lrGripperScrewerThreadPitchShow					:=	3;			
			VIS.lrGripperScrewerThreadTimesShow					:=	1.0;		
			VIS.nGripperScrewerCatchHeightSVShow				:=	110;
			VIS.bGripperScrewer1FindScrewShow					:=	FALSE;
			VIS.bGripperScrewer1Option4Show						:=	FALSE;
			VIS.lrGripperScrewer1FindingScrewDegreeShow			:=	260;
			VIS.bGripperScrewer1Option1Show						:=	FALSE;
			VIS.bGripperScrewer1Option2Show						:=	FALSE;
			VIS.bGripperScrewer1Option3Show						:=	TRUE;
			VIS.bGripperScrewer1Option5Show						:=	FALSE;
			VIS.bGripperScrewer1Option6Show						:=	TRUE;
			VIS.bGripperScrewer1Option7Show						:=	TRUE;
		ELSIF VIS.iPackageCapTypeShow	= 4 THEN // Typ nasadki (0-Fliptop, 1-Pompka/Atomizer, 2-Kulka, 3-Airless, 4-, 5- Deko, 6-Nakrętka_słoika
			;
		ELSIF VIS.iPackageCapTypeShow	= 5 THEN // Typ nasadki (0-Fliptop, 1-Pompka/Atomizer, 2-Kulka, 3-Airless, 4-, 5- Deko, 6-Nakrętka_słoika
			VIS.lrGripperScrewingTightTorqueShow				:=	0.5;
			VIS.lrGripperScrewing2TightTorqueShow				:=	0.5;
			VIS.iGripperScrewer1ToolShow						:=	3;//0-Dwu,1-Trój,2-Kształtowa/DoKulek,3-Wbijająca,4-Zasysająca
			VIS.lrGripperScrewer1VelocityShow					:=	90;
			VIS.nGripperScrewer1TightTimeShow					:=	300;
			VIS.lrGripperScrewerReadyPositionShow				:=	VIS.iPackageHeightShow + 60;	
			VIS.lrGripperScrewerPushingCapPositionShow			:=	VIS.iPackageHeightShow + 14;	
			VIS.lrGripperScrewerScrewingCapPositionShow			:=	VIS.iPackageHeightShow + 14;	
			VIS.lrGripperScrewerFindScrewPositionShow			:=	VIS.iPackageHeightShow + 14;
			VIS.lrGripperScrewerPressureShow					:=	30;
			VIS.lrGripperScrewerCatchPressureShow				:=	20;
			VIS.lrGripperScrewerPressureExhaustLevelShow		:=	100.0;
			VIS.lrGripperScrewerCatchPressureExhaustLevelShow	:=	100.0;
			VIS.lrGripperScrewerTurnoversToFullScrewedShow		:=	1;
			VIS.lrGripperScrewerThreadPitchShow					:=	3;			
			VIS.lrGripperScrewerThreadTimesShow					:=	1.0;		
			VIS.nGripperScrewerCatchHeightSVShow				:=	110;
			VIS.bGripperScrewer1FindScrewShow					:=	FALSE;
			VIS.bGripperScrewer1Option4Show						:=	FALSE;
			VIS.lrGripperScrewer1FindingScrewDegreeShow			:=	260;
			VIS.bGripperScrewer1Option1Show						:=	FALSE;
			VIS.bGripperScrewer1Option2Show						:=	FALSE;
			VIS.bGripperScrewer1Option3Show						:=	TRUE;
			VIS.bGripperScrewer1Option5Show						:=	FALSE;
			VIS.bGripperScrewer1Option6Show						:=	TRUE;
			VIS.bGripperScrewer1Option7Show						:=	TRUE;
		ELSIF VIS.iPackageCapTypeShow	= 6 THEN // Typ nasadki (0-Fliptop, 1-Pompka/Atomizer, 2-Kulka, 3-Airless, 4-, 5- Deko, 6-Nakrętka_słoika
			// Do wpisania słoik
			VIS.lrGripperScrewingTightTorqueShow				:=	0.5;
			VIS.lrGripperScrewing2TightTorqueShow				:=	0.5;
			VIS.iGripperScrewer1ToolShow						:=	1;//0-Dwu,1-Trój,2-Kształtowa/DoKulek,3-Wbijająca,4-Zasysająca
			VIS.lrGripperScrewer1VelocityShow					:=	90;
			VIS.nGripperScrewer1TightTimeShow					:=	300;
			VIS.lrGripperScrewerReadyPositionShow				:=	VIS.iPackageHeightShow + 60;	
			VIS.lrGripperScrewerPushingCapPositionShow			:=	VIS.iPackageHeightShow + 5;	
			VIS.lrGripperScrewerScrewingCapPositionShow			:=	VIS.iPackageHeightShow + 10;	
			VIS.lrGripperScrewerFindScrewPositionShow			:=	VIS.iPackageHeightShow + 10;	
			VIS.lrGripperScrewerPressureShow					:=	30;
			VIS.lrGripperScrewerCatchPressureShow				:=	20;
			VIS.lrGripperScrewerPressureExhaustLevelShow		:=	100.0;
			VIS.lrGripperScrewerCatchPressureExhaustLevelShow	:=	100.0;
			VIS.lrGripperScrewerTurnoversToFullScrewedShow		:=	1;
			VIS.lrGripperScrewerThreadPitchShow					:=	3;			
			VIS.lrGripperScrewerThreadTimesShow					:=	1.0;		
			VIS.nGripperScrewerCatchHeightSVShow				:=	110;
			VIS.bGripperScrewer1FindScrewShow					:=	FALSE;
			VIS.bGripperScrewer1Option4Show						:=	FALSE;
			VIS.lrGripperScrewer1FindingScrewDegreeShow			:=	260;
			VIS.bGripperScrewer1Option1Show						:=	FALSE;
			VIS.bGripperScrewer1Option2Show						:=	FALSE;
			VIS.bGripperScrewer1Option3Show						:=	TRUE;
			VIS.bGripperScrewer1Option5Show						:=	FALSE;
			VIS.bGripperScrewer1Option6Show						:=	TRUE;
			VIS.bGripperScrewer1Option7Show						:=	TRUE;
		END_IF
			
		//Test zakręcania		// Typ nasadki (0-Fliptop, 1-Pompka/Atomizer, 2-Kulka, 3-Airless, 4-, 5- Deko, 6-Nakrętka_słoika
		IF 		VIS.iPackageCapTypeShow	= 0 THEN 			VIS.lrCapCorrectCheckHeightPosSVShow 	:=	VIS.iPackageCappedHeightShow - 7;
		ELSIF 	VIS.iPackageCapTypeShow	= 1 THEN 			VIS.lrCapCorrectCheckHeightPosSVShow	:=	VIS.iPackageCappedHeightShow - 7;
		ELSIF 	VIS.iPackageCapTypeShow	= 2 THEN 			VIS.lrCapCorrectCheckHeightPosSVShow	:=	VIS.iPackageCappedHeightShow - 7;
		ELSIF 	VIS.iPackageCapTypeShow	= 3 THEN 			VIS.lrCapCorrectCheckHeightPosSVShow	:=	VIS.iPackageCappedHeightShow - 7;
		ELSIF 	VIS.iPackageCapTypeShow	= 4 THEN 			VIS.lrCapCorrectCheckHeightPosSVShow	:=	VIS.iPackageCappedHeightShow - 7;
		ELSIF 	VIS.iPackageCapTypeShow	= 5 THEN 			VIS.lrCapCorrectCheckHeightPosSVShow	:=	VIS.iPackageCappedHeightShow - 7;
		ELSIF 	VIS.iPackageCapTypeShow	= 6 THEN 			VIS.lrCapCorrectCheckHeightPosSVShow	:=	VIS.iPackageCappedHeightShow - 7;
		END_IF	
		
		//Robot
		//VIS.iBottleTransferPickOffsetZShow:=0; 		
		//VIS.iBottleTransferPick2OffsetZShow:=0;		
		VIS.iBottleTransferPlace1OffsetZShow				:=	-VIS.iPackagePuckInsertHeightShow; 	
		VIS.iBottleTransferPlace2OffsetZShow				:=	-VIS.iPackagePuckInsertHeightShow; 	
		//VIS.iBottleTransferSpeedShow:=90;			
		
		VIS.bRecipeCalculate := FALSE;
	END_IF
END_ACTION

ACTION aFactoryRecipes:
//VIS.sRecipeNameShow:='Factory Settings';
VIS.sRecipeIndexShow:='EAN_';
VIS.nRecipeIndexShow:=1;		
		
VIS.sRecipeDescriptionShow:="Pusto";
VIS.sRecipeDispencerDescriptionShow:=
"Dispensers:
-spouts: 16mm
-neck centering jaws: TK , TK";
VIS.sRecipeCapsDescriptionShow:=
"Caps:
-Crew head: 2-jaw. 3-jaw driving head
-Corner head jaw: TK
-Center clamp: TK
-Pack gripper jaws: TK , TtkmatK";
VIS.sRecipeFormersDescriptionShow:=
"Formers:
-Former insert: NONE, TK";
VIS.sRecipeRobotDescriptionShow:=
"Robot product:
-Open from center:
-Number of sets:1/2
-Type of feet: Large/Small";
VIS.sRecipeBottleSorterDescriptionShow:=
"Cap Feeder: Not Included";
VIS.sRecipeCapSorterDescriptionShow:=
"Bottle Feeder: Not Included";

VIS.iPackageCapTypeShow:= 0; 															//P030_Recipes.stRecipe.stUBL.iPackageCapTypeShow.diDefault		
VIS.iPackageCapDiameterShow:=20;		//srednica szyjki 								//  P030_Recipes.stRecipe.stUBL.		
				
VIS.bExEnableShow:=FALSE;																//	P030_Recipes.stRecipe.stUBL.	

VIS.bBottleFeederEnableShow:=FALSE;														//P030_Recipes.stRecipe.stUBL.
VIS.iBottleFeederTurntableVelocitySVShow:=900;											//P030_Recipes.stRecipe.stUBL.
VIS.iBottleFeederBottleSensorDelayShow:=100;											//P030_Recipes.stRecipe.stUBL.
VIS.iBottleFeederFormGateDelayShow:=200;												//P030_Recipes.stRecipe.stUBL.
VIS.iBottleFeederAllowFormDelayShow:=5000;												//P030_Recipes.stRecipe.stUBL.

VIS.bPucksInserterEnableShow:=FALSE;													//P030_Recipes.stRecipe.stUBL.
VIS.iPucksInserterTurntableVelocitySVShow:=900;											//P030_Recipes.stRecipe.stUBL.
VIS.iPucksInserterConveyorVelocitySVShow:=900;											//P030_Recipes.stRecipe.stUBL.
VIS.iPucksInserterBottleSensorDelayShow:=100;											//P030_Recipes.stRecipe.stUBL.
VIS.iPucksInserterFormGateDelayShow:=200;												//P030_Recipes.stRecipe.stUBL.
VIS.iPucksInserterAllowFormDelayShow:=1000;												//P030_Recipes.stRecipe.stUBL.
VIS.lrPucksInserterWheelOffsetShow:=3;													//P030_Recipes.stRecipe.stUBL.
VIS.lrPucksInserterWheelAccelerationShow:=2000;											//P030_Recipes.stRecipe.stUBL.	
VIS.lrPucksInserterWheelVelocityShow:=1600;                                             //P030_Recipes.stRecipe.stUBL.
VIS.lrPucksInserterHammerHeightSVShow:=285;                                             //P030_Recipes.stRecipe.stUBL.
//Vasyl 27.05 Stół podający	
VIS.udiPucksInserterPushTableVelocityShow			:=1000;								//P030_Recipes.stRecipe.stUBL.
VIS.iPucksInserterPushTableRollersVelocityShow    	:=1000;                             //P030_Recipes.stRecipe.stUBL.
VIS.udiPucksInserterPushTableActuatorPUSHDelayShow	:=3000;                             //P030_Recipes.stRecipe.stUBL.
VIS.udiPucksInserterPushTableActuatorPULLDelayShow	:=3000;                             //P030_Recipes.stRecipe.stUBL.
VIS.udiPucksInserterPushTableOFFDelayShow			:=3000;                             //P030_Recipes.stRecipe.stUBL.
VIS.bPucksInserterPushTableActuatorEnableShow	    :=FALSE;                            //P030_Recipes.stRecipe.stUBL.
VIS.bPucksInserterPushTableRollerEnableShow			:=FALSE;                            //P030_Recipes.stRecipe.stUBL.
VIS.bPucksInserterPushTableEnableShow			    :=FALSE;							//P030_Recipes.stRecipe.stUBL.


VIS.bGateBeforeDispencersEnableShow:=TRUE; 												//P030_Recipes.stRecipe.stUBL.
VIS.nGateBeforeDispencersTimeFormInsertingShow:=300;                                    //P030_Recipes.stRecipe.stUBL.
VIS.bGateAfterWeightEnableShow:=TRUE;                                                   //P030_Recipes.stRecipe.stUBL.
VIS.nGateAfterWeightTimeFormInsertingShow:=250;                                         //P030_Recipes.stRecipe.stUBL.
VIS.bGateRobotEnableShow:=TRUE;                                                         //P030_Recipes.stRecipe.stUBL.
VIS.nGateRobotTimeFormInsertingShow:=250;                                               //P030_Recipes.stRecipe.stUBL.
                                                                                        
VIS.bFormsDragingRightEnableShow:=TRUE;                                                //P030_Recipes.stRecipe.stUBL.
VIS.lrFormsDragingRightVelocityShow:=500;                                               //P030_Recipes.stRecipe.stUBL.
VIS.lrFormsDragingRightAccelerationShow:=2400;                                          //P030_Recipes.stRecipe.stUBL.
VIS.lrFormsDragingRightDecelerationShow:=2400;                                          //P030_Recipes.stRecipe.stUBL.
                                                                                        
VIS.bFormsDragingLeftEnableShow:=TRUE;	                                                //P030_Recipes.stRecipe.stUBL.
VIS.lrFormsDragingLeftVelocityShow:=500;                                                //P030_Recipes.stRecipe.stUBL.
VIS.lrFormsDragingLeftAccelerationShow:=2400;                                           //P030_Recipes.stRecipe.stUBL.
VIS.lrFormsDragingLeftDecelerationShow:=2400;                                           //P030_Recipes.stRecipe.stUBL.

VIS.bDosingTwoPhasesShow:= bTestDwuFaz;													//P030_Recipes.stRecipe.stUBL.
VIS.lrDispencersLifterReadyPositionShow:=280;                                           //P030_Recipes.stRecipe.stUBL.
VIS.uiDispencerStartDosingDelayShow:=500;                                               //P030_Recipes.stRecipe.stUBL.
VIS.bDispencer1EnableShow:=TRUE;                                                        //P030_Recipes.stRecipe.stUBL.
VIS.bDispencer2EnableShow:=TRUE;                                                        //P030_Recipes.stRecipe.stUBL.
VIS.bDispencer3EnableShow:=TRUE;                                                        //P030_Recipes.stRecipe.stUBL.
VIS.bDispencer4EnableShow:=TRUE;                                                        //P030_Recipes.stRecipe.stUBL.
                                                                                        
VIS.lrDispencer1DoseVolumeShow:=495;                                                    //P030_Recipes.stRecipe.stUBL.
VIS.lrDispencer1Phase1VolumeShow:=0;                                                    //P030_Recipes.stRecipe.stUBL.
VIS.lrDispencer1Phase2VolumeShow:=00;
VIS.lrDispencer1Phase1VelocityShow:=140;
VIS.lrDispencer1Phase2VelocityShow:=140;
VIS.lrDispencer1Phase3VelocityShow:=50;
VIS.lrDispencer1SuckVelocityShow:=300;
VIS.lrDispencer1Phase1AccelerationShow:=600;
VIS.lrDispencer1Phase2AccelerationShow:=400;
VIS.lrDispencer1Phase3AccelerationShow:=50;
VIS.lrDispencer1SuckAccelerationShow:=3000;
VIS.lrDispencer1Phase1DecelerationShow:=150;
VIS.lrDispencer1Phase2DecelerationShow:=2000;
VIS.lrDispencer1Phase3DecelerationShow:=50;
VIS.udiDispencer1DosingDoneDelayTimeShow:=300;
VIS.lrDispencer1SuckValveOpenVolumeShow:=0;
VIS.lrDispencer1SuckValveOpenTimeDelayShow:=0;
VIS.lrDispencer1SuckValveCloseVolumeShow:=0;
VIS.lrDispencer1SuckValveCloseTimeDelayShow:=0;
VIS.lrDispencer1DoseValveOpenVolumeShow:=0;
VIS.lrDispencer1DoseValveOpenTimeAccShow:=200;
VIS.lrDispencer1DoseValveCloseVolumeShow:=1;
VIS.lrDispencer1DoseValveCloseTimeDecShow:=0;
VIS.lrDispencer1DoseSuckingVolumeShow:=0;
VIS.lrDispencer1DoseSuckingTimeDelayShow:=0;
VIS.bDispencer1DoseSuckingShow:=FALSE;
VIS.bDispencer1LiftSynchroPh1Show:=FALSE;
VIS.bDispencer1LiftSynchroPh2Show:=TRUE;
VIS.bDispencer1LiftSynchroPh3Show:=TRUE;
VIS.lrDispencer1LifterStartDosePositionShow:=80;
VIS.lrDispencer1LifterStopDosePositionShow:=192;
VIS.lrDispencer1LifterVelocityShow:=1050;
VIS.lrDispencer1LifterAccelerationShow:=7000(*15000*);
VIS.lrDispencer1LifterDecelerationShow:=7000(*15000*);

VIS.lrDispencer2DoseVolumeShow:=260;
VIS.lrDispencer2Phase1VolumeShow:=0;
VIS.lrDispencer2Phase2VolumeShow:=0;
VIS.lrDispencer2Phase1VelocityShow:=140;
VIS.lrDispencer2Phase2VelocityShow:=240;
VIS.lrDispencer2Phase3VelocityShow:=50;
VIS.lrDispencer2SuckVelocityShow:=300;
VIS.lrDispencer2Phase1AccelerationShow:=600;
VIS.lrDispencer2Phase2AccelerationShow:=800;
VIS.lrDispencer2Phase3AccelerationShow:=50;
VIS.lrDispencer2SuckAccelerationShow:=3000;
VIS.lrDispencer2Phase1DecelerationShow:=150;
VIS.lrDispencer2Phase2DecelerationShow:=2000;
VIS.lrDispencer2Phase3DecelerationShow:=50;
VIS.udiDispencer2DosingDoneDelayTimeShow:=10;
VIS.lrDispencer2SuckValveOpenVolumeShow:=0;
VIS.lrDispencer2SuckValveOpenTimeDelayShow:=0;
VIS.lrDispencer2SuckValveCloseVolumeShow:=0;
VIS.lrDispencer2SuckValveCloseTimeDelayShow:=0;
VIS.lrDispencer2DoseValveOpenVolumeShow:=0;
VIS.lrDispencer2DoseValveOpenTimeAccShow:=200;
VIS.lrDispencer2DoseValveCloseVolumeShow:=1;
VIS.lrDispencer2DoseValveCloseTimeDecShow:=0;
VIS.lrDispencer2DoseSuckingVolumeShow:=0;
VIS.lrDispencer2DoseSuckingTimeDelayShow:=0;
VIS.bDispencer2DoseSuckingShow:=0;
VIS.bDispencer2LiftSynchroPh1Show:=FALSE;
VIS.bDispencer2LiftSynchroPh2Show:=TRUE;
VIS.bDispencer2LiftSynchroPh3Show:=FALSE;
VIS.lrDispencer2LifterStartDosePositionShow:=60;
VIS.lrDispencer2LifterStopDosePositionShow:=192;
VIS.lrDispencer2LifterVelocityShow:=1050;
VIS.lrDispencer2LifterAccelerationShow:=7000(*15000*);
VIS.lrDispencer2LifterDecelerationShow:=7000(*15000*);

VIS.bDispencersCatchEnableShow:=TRUE;
VIS.bDispencersCatchMaxPressureShow:=TRUE;
VIS.lrDispencersCatchHeightSVShow:=215;

VIS.lrDispencersCatch1ClosedValueShow:= 26.9;
VIS.lrDispencersCatch1OpenValueShow:= 61.3;
VIS.lrDispencersCatch2ClosedValueShow:= 21.6;
VIS.lrDispencersCatch2OpenValueShow:= 60;
VIS.lrDispencersCatch3ClosedValueShow:= 24;
VIS.lrDispencersCatch3OpenValueShow:= 63.3;
VIS.lrDispencersCatch4ClosedValueShow:= 19.8;
VIS.lrDispencersCatch4OpenValueShow:= 62.6;
VIS.lrDispencersCatchToleranceShow:= 15;

VIS.bTank1MixerEnableShow:=FALSE;
VIS.bTankHeatingEnableShow:=FALSE;											// Zezwolenie na pracę grzania
VIS.iTankHeatingTempSVShow:=60;
VIS.bTank1PressureEnableShow:=FALSE;
VIS.bTank1SupplyPumpEnableShow:=FALSE;
VIS.bTank2SupplyPumpEnableShow:=FALSE;
VIS.uTank1LevelSetpointShow:=90;
VIS.uTank2LevelSetpointShow:=90;
VIS.bTank1LevelSignalInvertShow:=FALSE;
VIS.bTank2LevelSignalInvertShow:=FALSE;

VIS.bWeight1EnableShow:=TRUE;
VIS.lrWeightMassSVShow:=495;
VIS.iWeight1ActuatorUpDelayShow:= 0;			//20;
VIS.iWeight2ActuatorUpDelayShow:= 0;			//20;
VIS.iWeight3ActuatorUpDelayShow:= 0;			//20;
VIS.iWeight4ActuatorUpDelayShow:= 0;			//20;
VIS.iWeight5ActuatorUpDelayShow:= 0;			//20;
VIS.iWeight6ActuatorUpDelayShow:= 0;			//20;

VIS.lrFormWeightShow:=0;
VIS.lrMass1DensityShow:=1;
VIS.lrMass2DensityShow:=1;
VIS.lrCupWeightShow:=0;
VIS.lrWholePackageWeightShow:=0;
VIS.lrWeight1MeasurmentCorrectionShow:=0;
VIS.bDispencer1WeightCorrectionEnableShow:=TRUE;
VIS.bDispencer2WeightCorrectionEnableShow:=TRUE;
VIS.bDispencer3WeightCorrectionEnableShow:=TRUE;
VIS.bDispencer4WeightCorrectionEnableShow:=TRUE;
VIS.lrWeightUpperToleranceShow:=1500;
VIS.lrWeightLowerToleranceShow:=1500;
VIS.iWeightCorrectionNumberOfSamplesShow:=2;

//Podajnik knotów                                  
VIS.bWickFeederEnableShow:=FALSE;
VIS.lrWickFeederHeightPosSVShow:=130;	
VIS.iWickFeederSorterTimeDelayOnShow:=1500;
VIS.iWickFeederSorterTimeDelayOffShow:=1500;
VIS.iWickFeederSorterTimeToEmptySleeveErrorShow:=300;	

				
//Przeciąganie podajnika knotów                 
VIS.bWickFeederDragingStationEnableShow:=FALSE;				
VIS.lrWickFeederDragingStationVelocityShow:=660;			
VIS.lrWickFeederDragingStationAccelerationShow:=2400;		
VIS.lrWickFeederDragingStationDecelerationShow:=2400;		

//Podajnik platynek
VIS.bLidFeederEnableShow:=FALSE;						
VIS.bLidFeederHeaterEnableShow:=FALSE;					
VIS.lrLidFeederHeightPosSVShow:=309;					
VIS.iLidFeederHeatingTimeShow:=200;							
VIS.iLidFeederTempHisteresisShow:=10;						
VIS.iLidFeeder1TempSVShow:=100;								
VIS.iLidFeeder2TempSVShow:=100;								

//Przeciąganie podajnika platynek
VIS.bLidFeederDragingStationEnableShow:=FALSE;			
VIS.lrLidFeederDragingStationVelocityShow:=500;		
VIS.lrLidFeederDragingStationAccelerationShow:=2400;		
VIS.lrLidFeederDragingStationDecelerationShow:=2400;		

//Sprawdzanie platynek
VIS.bLidPuttedCheckEnableShow:=FALSE;      				
VIS.lrLidPuttedCheckHeightSVShow:=200;  	 			
VIS.lrLidPuttedCheckPositionShow:=200; 				
VIS.lrLidPuttedCheckAreaShow:=200; 					
VIS.iLidPuttedCheckProgramShow:=0; 					

//Zgrzewanie
VIS.bLidSealerEnableShow:=FALSE;						
VIS.bLidSealerHeaterEnableShow:=FALSE;					
VIS.iLidSealerHeatingTimeShow:=200;					
VIS.lrLidSealerPressureShow:=100;					
VIS.lrLidSealerHeightPosSVShow:=285;				
VIS.iLidSealerTempHisteresisShow:=10;				
VIS.iLidSealer1TempSVShow:=100;				
VIS.iLidSealer2TempSVShow:=100;								

//ROPP
//Spowalniacz
VIS_ROPP.bROPPSlowerEnableShow					:=	FALSE;
VIS_ROPP.nROPPSlowerVelocitySVShow				:=	1800;                                
//Podajnik                     		
VIS_ROPP.bROPPFeederEnableShow					:=	FALSE;
VIS_ROPP.lrROPPFeederHeightPosSVShow			:=	200;
VIS_ROPP.iROPPFeederTimeDelayOnShow				:=	300;
VIS_ROPP.iROPPFeederTimeDelayOffShow			:=	300;
VIS_ROPP.iROPPFeederTimeToEmptySleeveErrorShow	:=	12200;                                 
//Przeciąganie                          
VIS_ROPP.bROPPDragEnableShow					:=	FALSE;
VIS_ROPP.lrROPPDragVelocityShow					:=	380;
VIS_ROPP.lrROPPDragAccelerationShow				:=	2400;
VIS_ROPP.lrROPPDragDecelerationShow				:=	2400;                             
//Zakrecanie                    		
VIS_ROPP.bROPPCappingEnableShow					:=	FALSE;
VIS_ROPP.lrROPPCappingHeightPosSVShow			:=	195;
VIS_ROPP.lrROPPCappingVelocitySVShow			:=	800;
VIS_ROPP.iROPPCappingTimeShow					:=	200;
VIS_ROPP.iROPPCappingTime2Show					:=	200;
VIS_ROPP.iROPPCapping1ToolShow					:=	1;

//Przeciąganie zgrzewania
VIS.bLidSealerDragingStationEnableShow:=FALSE;			
VIS.lrLidSealerDragingStationVelocityShow:=500;			
VIS.lrLidSealerDragingStationAccelerationShow:=2400;	
VIS.lrLidSealerDragingStationDecelerationShow:=2400;	

VIS.bCapFeederGateEnableShow:=FALSE;			
VIS.iCapFeederGateBlockingTimeShow:=100;
                      				
VIS.bCapFeederEnableShow:=FALSE;					
VIS.lrCapFeederHeightPosSVShow:=205.4;			
VIS.iCapFeederTimeDelayOnShow:=1000;
VIS.iCapFeederTimeDelayOffShow:=100;
VIS.iCapFeederTimeToEmptySleeveErrorShow:=30;

VIS.bCapSorterDragEnableShow:=TRUE;
VIS.lrCapSorterDragVelocityShow:=380;
VIS.lrCapSorterDragAccelerationShow:=2400;
VIS.lrCapSorterDragDecelerationShow:=2400;

VIS.bCapPuttedCheckEnableShow:=TRUE;
VIS.lrCapPuttedCheckHeightPosSVShow:= 203;

VIS.bGripperScrewer1EnableShow:=TRUE;
VIS.lrGripperScrewingTightTorqueShow:=0.8;
VIS.bGripperScrewer2EnableShow:=TRUE;
VIS.lrGripperScrewing2TightTorqueShow:=1.1;
VIS.iGripperScrewer1ToolShow:=0;
VIS.lrGripperScrewer1VelocityShow:=90;
VIS.nGripperScrewer1TightTimeShow:=100;
VIS.iGripperScrewer1StartDelayShow:=0;
VIS.lrGripperScrewerReadyPositionShow:=	P10_GripperScrewer.fb2GripperScrewer1.lrMaxHeightPosition - 10;
VIS.lrGripperScrewerPushingCapPositionShow:=P10_GripperScrewer.fb2GripperScrewer1.lrMaxHeightPosition - 20;
VIS.lrGripperScrewerScrewingCapPositionShow:=P10_GripperScrewer.fb2GripperScrewer1.lrMaxHeightPosition - 20;
VIS.lrGripperScrewerFindScrewPositionShow:=P10_GripperScrewer.fb2GripperScrewer1.lrMaxHeightPosition - 20;
VIS.lrGripperScrewerPressureShow:=40;
VIS.lrGripperScrewerCatchPressureShow:=20;
VIS.lrGripperScrewerPressureExhaustLevelShow:= 100.0;
VIS.lrGripperScrewerCatchPressureExhaustLevelShow:= 100.0;
VIS.lrGripperScrewerTurnoversToFullScrewedShow:=0.5;
VIS.lrGripperScrewerThreadPitchShow:=0.5;			
VIS.lrGripperScrewerThreadTimesShow:=1.0;		
VIS.nGripperScrewerCatchHeightSVShow:= 160;
VIS.bGripperScrewer1FindScrewShow:=TRUE;
VIS.bGripperScrewer1Option4Show:=FALSE;
VIS.lrGripperScrewer1FindingScrewDegreeShow:=260;
VIS.bGripperScrewer1Option1Show:=FALSE;
VIS.bGripperScrewer1Option2Show:=FALSE;
VIS.bGripperScrewer1Option3Show:=TRUE;
VIS.bGripperScrewer1Option5Show:=FALSE;
VIS.bGripperScrewer1Option6Show:=FALSE;
VIS.bGripperScrewer1Option7Show:=TRUE;

VIS.bBottleDragingStationEnableShow:=TRUE;
VIS.lrBottleDragingStationVelocityShow:=380;

VIS.bCapCorrectCheckEnableShow:=TRUE;
VIS.lrCapCorrectCheckHeightPosSVShow:=200.5;

VIS.bBottleTransferEnableShow:=TRUE;   //było true
VIS.nBottleTransferProgramShow:=0;
VIS.iBottleTransferPickOffsetXShow:=0; 		
VIS.iBottleTransferPickOffsetYShow:=0; 		
VIS.iBottleTransferPickOffsetZShow:=0; 		
VIS.iBottleTransferPick2OffsetXShow:=0;		
VIS.iBottleTransferPick2OffsetYShow:=0;		
VIS.iBottleTransferPick2OffsetZShow:=0;		
VIS.iBottleTransferPlace1OffsetXShow:=0; 	
VIS.iBottleTransferPlace1OffsetYShow:=0; 	
VIS.iBottleTransferPlace1OffsetZShow:=0; 	
VIS.iBottleTransferPlace2OffsetXShow:=0; 	
VIS.iBottleTransferPlace2OffsetYShow:=0;	
VIS.iBottleTransferPlace2OffsetZShow:=0; 	
VIS.iBottleTransferSpeedShow:=30;			
VIS.bBottleTransferInkJetEnableShow:=FALSE;	
VIS.bBottleTransferPickOnlyOneShow:=FALSE;		

VIS.bBottleTransferAfterDragEnableShow:=TRUE;

VIS.bBadBottleConveyorEnableShow:=TRUE;
VIS.nBadBottleConveyorVelocitySVShow:=1300;

VIS.bLabelMachineEnableShow:=FALSE;

VIS.bExitTurnTable1EnableShow:=FALSE;
VIS.bExitConveyorEnableShow:=FALSE;
VIS.nExitConveyorVelocitySVShow := 700;

VIS.bFormTransportersEnableShow:=TRUE;
VIS.nFormTransportersDispencerVelocitySVShow:=1200;
VIS.nFormTransportersScrewerVelocitySVShow:=1200;
VIS.nFormTransportersAfterCapSorterVelocitySVShow:=1200;
VIS.nFormTransportersBeforeScrewerVelocitySVShow:=1100;
VIS.nFormTransportersSlowerVelocitySVShow:= 1800;
VIS.nFormTransportersAfterScrewerVelocitySVShow:=1100;


VIS.bCircularInkjetEnableShow:=FALSE;	
VIS.iCircularInkjetSpeedShow:=1200;	
VIS.iCircularInkjetDelayShow:=200;	
VIS.iCircularInkjetHoldShow:=300;
END_ACTION

ACTION aLimits:
(*
Nazwa:			aLimits
Wersja:			v0.1 			
Autor:			DP
Urzadzenia:		
Konfiguracja:	
Info:
-  blokany nastaw w recepturach które się wykluczają
Uwagi:
- 
Zmiany:

*)
(*WŁĄCZONE SŁOIKI*)

IF VIS.nExitConveyorVelocitySVShow < 100 THEN
	VIS.nExitConveyorVelocitySVShow := 900;
END_IF
END_ACTION

ACTION aShowToAll:
sRecipeName:=WSTRING_TO_STRING(VIS.sRecipeNameShow);
sRecipeIndex:=VIS.sRecipeIndexShow;		
nRecipeIndex:=VIS.nRecipeIndexShow;		
																			
iPackageCapType:=VIS.iPackageCapTypeShow;	
iPackageCapDiameter:=VIS.iPackageCapDiameterShow;
															
//bExEnable:=VIS.bExEnableShow;
VIS.bExEnableShow;
bExEnable:=GVL_IO.IbExModeSwitchExMode AND NOT GVL_IO.IbExModeSwitchNormalMode;
															
bBottleFeederEnable:= VIS.bBottleFeederEnableShow;
iBottleFeederTurntableVelocitySV:=VIS.iBottleFeederTurntableVelocitySVShow;
iBottleFeederBottleSensorDelay:=VIS.iBottleFeederBottleSensorDelayShow;
iBottleFeederFormGateDelay:=VIS.iBottleFeederFormGateDelayShow;
iBottleFeederAllowFormDelay:=VIS.iBottleFeederAllowFormDelayShow;
															
bPucksInserterEnable:=VIS.bPucksInserterEnableShow;
iPucksInserterTurntableVelocitySV:=VIS.iPucksInserterTurntableVelocitySVShow;
iPucksInserterConveyorVelocitySV:=VIS.iPucksInserterConveyorVelocitySVShow;
iPucksInserterBottleSensorDelay:=VIS.iPucksInserterBottleSensorDelayShow;
iPucksInserterFormGateDelay:=VIS.iPucksInserterFormGateDelayShow;
iPucksInserterAllowFormDelay:=VIS.iPucksInserterAllowFormDelayShow;
lrPucksInserterWheelOffset:=VIS.lrPucksInserterWheelOffsetShow;	
lrPucksInserterWheelAcceleration:=VIS.lrPucksInserterWheelAccelerationShow;
lrPucksInserterWheelVelocity:=VIS.lrPucksInserterWheelVelocityShow;	
lrPucksInserterHammerHeightSV:=VIS.lrPucksInserterHammerHeightSVShow;

//Vasyl 27.05 Stół podający
udiPucksInserterPushTable_m1_VelocitySV:=VIS.udiPucksInserterPushTableVelocityShow;		
udiPucksInserterPushTable_m3_VelocitySV:=VIS.udiPucksInserterPushTableVelocityShow+500;		
udiPucksInserterPushTable_m2_VelocitySV:=VIS.iPucksInserterPushTableRollersVelocityShow;
	
udiPucksInserterPushTableActuatorPUSHDelay:=VIS.udiPucksInserterPushTableActuatorPUSHDelayShow;
udiPucksInserterPushTableActuatorPULLDelay:=VIS.udiPucksInserterPushTableActuatorPULLDelayShow;
udiPucksInserterPushTableOFFDelay	:= VIS.udiPucksInserterPushTableOFFDelayShow;
bPucksInserterPushTable_m2_Enable	 :=VIS.bPucksInserterPushTableRollerEnableShow;		
bPucksInserterPushTable_m1_Enable	 :=VIS.bPucksInserterPushTableEnableShow;
bPucksInserterPushTable_m3_Enable	 :=VIS.bPucksInserterPushTableEnableShow;			


VIS.bGateBeforeDispencersEnableShow := TRUE; (*wizka kasuje*)
bGateBeforeDispencersEnable:=VIS.bGateBeforeDispencersEnableShow;
nGateBeforeDispencersTimeFormInserting:=VIS.nGateBeforeDispencersTimeFormInsertingShow;
VIS.bGateAfterWeightEnableShow := TRUE;(*wizka kasuje*)
bGateAfterWeightEnable:=VIS.bGateAfterWeightEnableShow;
nGateAfterWeightTimeFormInserting:=VIS.nGateAfterWeightTimeFormInsertingShow;
VIS.bGateRobotEnableShow := TRUE;(*wizka kasuje*)
bGateRobotEnable:=VIS.bGateRobotEnableShow;
nGateRobotTimeFormInserting:=VIS.nGateRobotTimeFormInsertingShow;
															
bFormsDragingRightEnable:=VIS.bFormsDragingRightEnableShow;
lrFormsDragingRightVelocity:=VIS.lrFormsDragingRightVelocityShow;
lrFormsDragingRightAcceleration:=VIS.lrFormsDragingRightAccelerationShow;
lrFormsDragingRightDeceleration:=VIS.lrFormsDragingRightDecelerationShow;
															
bFormsDragingLeftEnable:=VIS.bFormsDragingLeftEnableShow;	
lrFormsDragingLeftVelocity:=VIS.lrFormsDragingLeftVelocityShow;
lrFormsDragingLeftAcceleration:=VIS.lrFormsDragingLeftAccelerationShow;
lrFormsDragingLeftDeceleration:=VIS.lrFormsDragingLeftDecelerationShow;
//IF bDosingTwoPhases THEN
//	VIS.lrFormsDragingLeftDecelerationShow := 400;
//END_IF
															
//bDosingTwoPhases:=VIS.bDosingTwoPhasesShow;
VIS.bDosingTwoPhasesShow;
lrDispencersLifterReadyPosition:=VIS.lrDispencersLifterReadyPositionShow;
uiDispencerStartDosingDelay:=VIS.uiDispencerStartDosingDelayShow;
bDispencer1Enable:=VIS.bDispencer1EnableShow;
bDispencer2Enable:=VIS.bDispencer2EnableShow;
bDispencer3Enable:=VIS.bDispencer3EnableShow;
bDispencer4Enable:=VIS.bDispencer4EnableShow;
															
lrDispencer1DoseVolume:=VIS.lrDispencer1DoseVolumeShow;
lrDispencer1Phase1Volume:=VIS.lrDispencer1Phase1VolumeShow;
lrDispencer1Phase2Volume:=VIS.lrDispencer1Phase2VolumeShow;
lrDispencer1Phase1Velocity:=VIS.lrDispencer1Phase1VelocityShow;
lrDispencer1Phase2Velocity:=VIS.lrDispencer1Phase2VelocityShow;
lrDispencer1Phase3Velocity:=VIS.lrDispencer1Phase3VelocityShow;
lrDispencer1SuckVelocity:=VIS.lrDispencer1SuckVelocityShow;
lrDispencer1Phase1Acceleration:=VIS.lrDispencer1Phase1AccelerationShow;
lrDispencer1Phase2Acceleration:=VIS.lrDispencer1Phase2AccelerationShow;
lrDispencer1Phase3Acceleration:=VIS.lrDispencer1Phase3AccelerationShow;
lrDispencer1SuckAcceleration:=VIS.lrDispencer1SuckAccelerationShow;
lrDispencer1Phase1Deceleration:=VIS.lrDispencer1Phase1DecelerationShow;
lrDispencer1Phase2Deceleration:=VIS.lrDispencer1Phase2DecelerationShow;
lrDispencer1Phase3Deceleration:=VIS.lrDispencer1Phase3DecelerationShow;
udiDispencer1DosingDoneDelayTime:=VIS.udiDispencer1DosingDoneDelayTimeShow;
lrDispencer1SuckValveOpenVolume:=VIS.lrDispencer1SuckValveOpenVolumeShow;
lrDispencer1SuckValveOpenTimeDelay:=VIS.lrDispencer1SuckValveOpenTimeDelayShow;
lrDispencer1SuckValveCloseVolume:=VIS.lrDispencer1SuckValveCloseVolumeShow;
lrDispencer1SuckValveCloseTimeDelay:=VIS.lrDispencer1SuckValveCloseTimeDelayShow;
lrDispencer1DoseValveOpenVolume:=VIS.lrDispencer1DoseValveOpenVolumeShow;
lrDispencer1DoseValveOpenTimeAcc:=VIS.lrDispencer1DoseValveOpenTimeAccShow;
lrDispencer1DoseValveCloseVolume:=VIS.lrDispencer1DoseValveCloseVolumeShow;
lrDispencer1DoseValveCloseTimeDec:=VIS.lrDispencer1DoseValveCloseTimeDecShow;
lrDispencer1DoseSuckingVolume:=VIS.lrDispencer1DoseSuckingVolumeShow;
lrDispencer1DoseSuckingTimeDelay:=VIS.lrDispencer1DoseSuckingTimeDelayShow;
bDispencer1DoseSucking:=VIS.bDispencer1DoseSuckingShow;
bDispencer1LiftSynchroPh1:=VIS.bDispencer1LiftSynchroPh1Show;
bDispencer1LiftSynchroPh2:=VIS.bDispencer1LiftSynchroPh2Show;
bDispencer1LiftSynchroPh3:=VIS.bDispencer1LiftSynchroPh3Show;
lrDispencer1LifterStartDosePosition:=VIS.lrDispencer1LifterStartDosePositionShow;
lrDispencer1LifterStopDosePosition:=VIS.lrDispencer1LifterStopDosePositionShow;
lrDispencer1LifterVelocity:=VIS.lrDispencer1LifterVelocityShow:=1050;
lrDispencer1LifterAcceleration:=VIS.lrDispencer1LifterAccelerationShow;
lrDispencer1LifterDeceleration:=VIS.lrDispencer1LifterDecelerationShow;
															
lrDispencer2DoseVolume:=VIS.lrDispencer2DoseVolumeShow;
lrDispencer2Phase1Volume:=VIS.lrDispencer2Phase1VolumeShow;
lrDispencer2Phase2Volume:=VIS.lrDispencer2Phase2VolumeShow;
lrDispencer2Phase1Velocity:=VIS.lrDispencer2Phase1VelocityShow;
lrDispencer2Phase2Velocity:=VIS.lrDispencer2Phase2VelocityShow;
lrDispencer2Phase3Velocity:=VIS.lrDispencer2Phase3VelocityShow;
lrDispencer2SuckVelocity:=VIS.lrDispencer2SuckVelocityShow;
lrDispencer2Phase1Acceleration:=VIS.lrDispencer2Phase1AccelerationShow;
lrDispencer2Phase2Acceleration:=VIS.lrDispencer2Phase2AccelerationShow;
lrDispencer2Phase3Acceleration:=VIS.lrDispencer2Phase3AccelerationShow;
lrDispencer2SuckAcceleration:=VIS.lrDispencer2SuckAccelerationShow;
lrDispencer2Phase1Deceleration:=VIS.lrDispencer2Phase1DecelerationShow;
lrDispencer2Phase2Deceleration:=VIS.lrDispencer2Phase2DecelerationShow;
lrDispencer2Phase3Deceleration:=VIS.lrDispencer2Phase3DecelerationShow;
udiDispencer2DosingDoneDelayTime:=VIS.udiDispencer2DosingDoneDelayTimeShow;
lrDispencer2SuckValveOpenVolume:=VIS.lrDispencer2SuckValveOpenVolumeShow;
lrDispencer2SuckValveOpenTimeDelay:=VIS.lrDispencer2SuckValveOpenTimeDelayShow;
lrDispencer2SuckValveCloseVolume:=VIS.lrDispencer2SuckValveCloseVolumeShow;
lrDispencer2SuckValveCloseTimeDelay:=VIS.lrDispencer2SuckValveCloseTimeDelayShow;
lrDispencer2DoseValveOpenVolume:=VIS.lrDispencer2DoseValveOpenVolumeShow;
lrDispencer2DoseValveOpenTimeAcc:=VIS.lrDispencer2DoseValveOpenTimeAccShow;
lrDispencer2DoseValveCloseVolume:=VIS.lrDispencer2DoseValveCloseVolumeShow;
lrDispencer2DoseValveCloseTimeDec:=VIS.lrDispencer2DoseValveCloseTimeDecShow;
lrDispencer2DoseSuckingVolume:=VIS.lrDispencer2DoseSuckingVolumeShow;
lrDispencer2DoseSuckingTimeDelay:=VIS.lrDispencer2DoseSuckingTimeDelayShow;
bDispencer2DoseSucking:=VIS.bDispencer2DoseSuckingShow;
bDispencer2LiftSynchroPh1:=VIS.bDispencer2LiftSynchroPh1Show;
bDispencer2LiftSynchroPh2:=VIS.bDispencer2LiftSynchroPh2Show;
bDispencer2LiftSynchroPh3:=VIS.bDispencer2LiftSynchroPh3Show;
lrDispencer2LifterStartDosePosition:=VIS.lrDispencer2LifterStartDosePositionShow;
lrDispencer2LifterStopDosePosition:=VIS.lrDispencer2LifterStopDosePositionShow;
lrDispencer2LifterVelocity:=VIS.lrDispencer2LifterVelocityShow:=1050;
lrDispencer2LifterAcceleration:=VIS.lrDispencer2LifterAccelerationShow;
lrDispencer2LifterDeceleration:=VIS.lrDispencer2LifterDecelerationShow;
															
bDispencersCatchEnable:=VIS.bDispencersCatchEnableShow;
bDispencersCatchMaxPressure:=VIS.bDispencersCatchMaxPressureShow;
lrDispencersCatchHeightSV:=VIS.lrDispencersCatchHeightSVShow;
															
lrDispencersCatch1ClosedValue:=VIS.lrDispencersCatch1ClosedValueShow;
lrDispencersCatch1OpenValue:=VIS.lrDispencersCatch1OpenValueShow;
lrDispencersCatch2ClosedValue:=VIS.lrDispencersCatch2ClosedValueShow;
lrDispencersCatch2OpenValue:=VIS.lrDispencersCatch2OpenValueShow;
lrDispencersCatch3ClosedValue:=VIS.lrDispencersCatch3ClosedValueShow;
lrDispencersCatch3OpenValue:=VIS.lrDispencersCatch3OpenValueShow;
lrDispencersCatch4ClosedValue:=VIS.lrDispencersCatch4ClosedValueShow;
lrDispencersCatch4OpenValue:=VIS.lrDispencersCatch4OpenValueShow;
lrDispencersCatchTolerance:=VIS.lrDispencersCatchToleranceShow;
															
bTank1MixerEnable:=VIS.bTank1MixerEnableShow;
bTankHeatingEnable:=VIS.bTankHeatingEnableShow;
iTankHeatingTempSV:=VIS.iTankHeatingTempSVShow;
bTank1PressureEnable:=VIS.bTank1PressureEnableShow;
bTank1SupplyPumpEnable:=VIS.bTank1SupplyPumpEnableShow;
bTank2SupplyPumpEnable:=VIS.bTank2SupplyPumpEnableShow;
uTank1LevelSetpoint:=VIS.uTank1LevelSetpointShow;
uTank2LevelSetpoint:=VIS.uTank2LevelSetpointShow;
bTank1LevelSignalInvert:=VIS.bTank1LevelSignalInvertShow;
bTank2LevelSignalInvert:=VIS.bTank2LevelSignalInvertShow;
bTankRainbowMode:=VIS.bTankRainbowModeShow;														
bWeight1Enable:=VIS.bWeight1EnableShow;
bWeightLiftEnable:=VIS.bWeight1EnableShow;
lrWeightMassSV:=VIS.lrWeightMassSVShow;
iWeight1ActuatorUpDelay:=VIS.iWeight1ActuatorUpDelayShow;
iWeight2ActuatorUpDelay:=VIS.iWeight2ActuatorUpDelayShow;
iWeight3ActuatorUpDelay:=VIS.iWeight3ActuatorUpDelayShow;
iWeight4ActuatorUpDelay:=VIS.iWeight4ActuatorUpDelayShow;

VIS.iWeight5ActuatorUpDelayShow:=30;
VIS.iWeight6ActuatorUpDelayShow:=30;
iWeight5ActuatorUpDelay:=VIS.iWeight5ActuatorUpDelayShow;
iWeight6ActuatorUpDelay:=VIS.iWeight6ActuatorUpDelayShow;
															
lrFormWeight:=VIS.lrFormWeightShow;
lrMass1Density:=VIS.lrMass1DensityShow;
lrMass2Density:=VIS.lrMass2DensityShow;
lrCupWeight:=VIS.lrCupWeightShow;
lrWholePackageWeight:=VIS.lrWholePackageWeightShow;
lrWeight1MeasurmentCorrection:=VIS.lrWeight1MeasurmentCorrectionShow;
bDispencer1WeightCorrectionEnable:=VIS.bDispencer1WeightCorrectionEnableShow;
bDispencer2WeightCorrectionEnable:=VIS.bDispencer2WeightCorrectionEnableShow;
bDispencer3WeightCorrectionEnable:=VIS.bDispencer3WeightCorrectionEnableShow;
bDispencer4WeightCorrectionEnable:=VIS.bDispencer4WeightCorrectionEnableShow;
lrWeightUpperTolerance:=VIS.lrWeightUpperToleranceShow;
lrWeightLowerTolerance:=VIS.lrWeightLowerToleranceShow;
iWeightCorrectionNumberOfSamples:=VIS.iWeightCorrectionNumberOfSamplesShow;

//Podajnik knotów                   
bWickFeederEnable:=VIS.bWickFeederEnableShow;						
lrWickFeederHeightPosSV:=VIS.lrWickFeederHeightPosSVShow;					
iWickFeederSorterTimeDelayOn:=VIS.iWickFeederSorterTimeDelayOnShow;
iWickFeederSorterTimeDelayOff:=VIS.iWickFeederSorterTimeDelayOffShow;
iWickFeederSorterTimeToEmptySleeveError:=VIS.iWickFeederSorterTimeToEmptySleeveErrorShow;	
                                             
//Przeciąganie podajnika knotów             
bWickFeederDragingStationEnable:=VIS.bWickFeederDragingStationEnableShow OR VIS.bWickFeederEnableShow;			
lrWickFeederDragingStationVelocity:=VIS.lrWickFeederDragingStationVelocityShow;	
lrWickFeederDragingStationAcceleration:=VIS.lrWickFeederDragingStationAccelerationShow;	
lrWickFeederDragingStationDeceleration:=VIS.lrWickFeederDragingStationDecelerationShow;	

		
//Podajnik platynek
bLidFeederEnable := VIS.bLidFeederEnableShow;						
bLidFeederHeaterEnable := VIS.bLidFeederHeaterEnableShow;					
lrLidFeederHeightPosSV := VIS.lrLidFeederHeightPosSVShow;				
iLidFeederHeatingTime := VIS.iLidFeederHeatingTimeShow;					
iLidFeederTempHisteresis := VIS.iLidFeederTempHisteresisShow;						
iLidFeeder1TempSV := VIS.iLidFeeder1TempSVShow;							
iLidFeeder2TempSV := VIS.iLidFeeder2TempSVShow;							
                                                    
//Przeciąganie podajnika platynek
//VIS.bLidFeederDragingStationEnableShow :=	VIS.bLidFeederEnableShow;
bLidFeederDragingStationEnable := VIS.bLidFeederDragingStationEnableShow;			
lrLidFeederDragingStationVelocity := VIS.lrLidFeederDragingStationVelocityShow;	
lrLidFeederDragingStationAcceleration := VIS.lrLidFeederDragingStationAccelerationShow;		
lrLidFeederDragingStationDeceleration := VIS.lrLidFeederDragingStationDecelerationShow;	
                                                    
//Sprawdzanie platynek
bLidPuttedCheckEnable := VIS.bLidPuttedCheckEnableShow;   				
lrLidPuttedCheckHeightSV := VIS.lrLidPuttedCheckHeightSVShow; 			
lrLidPuttedCheckPosition := VIS.lrLidPuttedCheckPositionShow;			
lrLidPuttedCheckArea := VIS.lrLidPuttedCheckAreaShow;					
iLidPuttedCheckProgram := VIS.iLidPuttedCheckProgramShow; 					
                                                    
//Zgrzewanie
bLidSealerEnable := VIS.bLidSealerEnableShow;						
bLidSealerHeaterEnable := VIS.bLidSealerHeaterEnableShow;				
iLidSealerHeatingTime := VIS.iLidSealerHeatingTimeShow;				
lrLidSealerPressure := VIS.lrLidSealerPressureShow;			
lrLidSealerHeightPosSV := VIS.lrLidSealerHeightPosSVShow;				
iLidSealerTempHisteresis := VIS.iLidSealerTempHisteresisShow;				
iLidSealer1TempSV := VIS.iLidSealer1TempSVShow;				
iLidSealer2TempSV := VIS.iLidSealer2TempSVShow;							
 
//ROPP
//Spowalniacz
bROPPSlowerEnable:= VIS_ROPP.bROPPSlowerEnableShow;

IF NOT P00_PackML.bROPPDelayAfterStartFullRegister THEN
   nROPPSlowerVelocitySV	:=	700;
ELSE
    nROPPSlowerVelocitySV:=VIS_ROPP.nROPPSlowerVelocitySVShow;  
END_IF                       
//Podajnik                     		
bROPPFeederEnable:=VIS_ROPP.bROPPFeederEnableShow;
lrROPPFeederHeightPosSV:=VIS_ROPP.lrROPPFeederHeightPosSVShow;
iROPPFeederTimeDelayOn:=VIS_ROPP.iROPPFeederTimeDelayOnShow;
iROPPFeederTimeDelayOff:=VIS_ROPP.iROPPFeederTimeDelayOffShow;
iROPPFeederTimeToEmptySleeveError:=VIS_ROPP.iROPPFeederTimeToEmptySleeveErrorShow;                                  
//Przeciąganie                          
bROPPDragEnable:=VIS_ROPP.bROPPDragEnableShow;
lrROPPDragVelocity:=VIS_ROPP.lrROPPDragVelocityShow;
lrROPPDragAcceleration:=VIS_ROPP.lrROPPDragAccelerationShow;
lrROPPDragDeceleration:=VIS_ROPP.lrROPPDragDecelerationShow;                               
//Zakrecanie                    		
bROPPCappingEnable:=VIS_ROPP.bROPPCappingEnableShow;
lrROPPCappingHeightPosSV:=VIS_ROPP.lrROPPCappingHeightPosSVShow;
lrROPPCappingVelocitySV:=VIS_ROPP.lrROPPCappingVelocitySVShow;
iROPPCappingTime:=VIS_ROPP.iROPPCappingTimeShow;
iROPPCappingTime2:=VIS_ROPP.iROPPCappingTime2Show;
iROPPCapping1Tool:=VIS_ROPP.iROPPCapping1ToolShow;

                                                
//Przeciąganie zgrzewania
VIS.bLidSealerDragingStationEnableShow :=VIS.bLidSealerEnableShow OR VIS.bDosingTwoPhasesShow OR 
										P00_PackML.tofbDosingTwoPhases.Q OR VIS.bLidSealerDragingStationEnableShow OR
										bWickFeederEnable;
bLidSealerDragingStationEnable := VIS.bLidSealerDragingStationEnableShow;			
lrLidSealerDragingStationVelocity := VIS.lrLidSealerDragingStationVelocityShow;		
lrLidSealerDragingStationAcceleration := VIS.lrLidSealerDragingStationAccelerationShow;	
lrLidSealerDragingStationDeceleration := VIS.lrLidSealerDragingStationDecelerationShow;
												
bCapFeederGateEnable:=VIS.bCapFeederGateEnableShow;		
iCapFeederGateBlockingTime:=VIS.iCapFeederGateBlockingTimeShow;
                  																				                      				
bCapFeederEnable:=VIS.bCapFeederEnableShow;						
lrCapFeederHeightPosSV:=VIS.lrCapFeederHeightPosSVShow;			
iCapFeederTimeDelayOn:=VIS.iCapFeederTimeDelayOnShow;
iCapFeederTimeDelayOff:=VIS.iCapFeederTimeDelayOffShow;
iCapFeederTimeToEmptySleeveError:=VIS.iCapFeederTimeToEmptySleeveErrorShow;

bCapSorterOnlyWeightOKEnable:=VIS.bCapSorterOnlyWeightOKEnableShow;

bCapSorterDragEnable:=VIS.bCapSorterDragEnableShow;
lrCapSorterDragVelocity:=VIS.lrCapSorterDragVelocityShow;
lrCapSorterDragAcceleration:=VIS.lrCapSorterDragAccelerationShow;
lrCapSorterDragDeceleration:=VIS.lrCapSorterDragDecelerationShow;

VIS.bWenglorSensorCapPuttedShow := TRUE;
													
bCapPuttedCheckEnable:=VIS.bCapPuttedCheckEnableShow;
lrCapPuttedCheckHeightPosSV:=VIS.lrCapPuttedCheckHeightPosSVShow;
															
bGripperScrewer1Enable:=VIS.bGripperScrewer1EnableShow;
lrGripperScrewingTightTorque:=VIS.lrGripperScrewingTightTorqueShow;
bGripperScrewer2Enable:=VIS.bGripperScrewer2EnableShow;
lrGripperScrewing2TightTorque:=VIS.lrGripperScrewing2TightTorqueShow;
iGripperScrewer1Tool:=VIS.iGripperScrewer1ToolShow;
lrGripperScrewerVelocity:=VIS.lrGripperScrewer1VelocityShow;
nGripperScrewerTightTime:=VIS.nGripperScrewer1TightTimeShow;
iGripperScrewerStartDelay:=VIS.iGripperScrewer1StartDelayShow;
lrGripperScrewerReadyPosition:=VIS.lrGripperScrewerReadyPositionShow;
lrGripperScrewerPushingCapPosition:=VIS.lrGripperScrewerPushingCapPositionShow;
lrGripperScrewerScrewingCapPosition:=VIS.lrGripperScrewerScrewingCapPositionShow;
lrGripperScrewerFindScrewPosition:=VIS.lrGripperScrewerFindScrewPositionShow;
lrGripperScrewerPressure:=VIS.lrGripperScrewerPressureShow;
lrDispencerCatchPressure:=VIS.lrDispencerCatchPressureShow;
lrGripperScrewerCatchPressure:=VIS.lrGripperScrewerCatchPressureShow;
lrGripperScrewerPressureExhaustLevel:=VIS.lrGripperScrewerPressureExhaustLevelShow:=100;
lrGripperScrewerCatchPressureExhaustLevel:=VIS.lrGripperScrewerCatchPressureExhaustLevelShow:=100;
lrGripperScrewerTurnoversToFullScrewed:=VIS.lrGripperScrewerTurnoversToFullScrewedShow;
lrGripperScrewerThreadPitch:=VIS.lrGripperScrewerThreadPitchShow;			
lrGripperScrewerThreadTimes:=VIS.lrGripperScrewerThreadTimesShow;	
nGripperScrewerCatchHeightSV:=VIS.nGripperScrewerCatchHeightSVShow;
bGripperScrewerFindScrew:=VIS.bGripperScrewer1FindScrewShow;
bGripperScrewerOption4:=VIS.bGripperScrewer1Option4Show;
lrGripperScrewerFindingScrewDegree:=VIS.lrGripperScrewer1FindingScrewDegreeShow;
bGripperScrewerOption1:=VIS.bGripperScrewer1Option1Show;
bGripperScrewerOption2:=VIS.bGripperScrewer1Option2Show;
bGripperScrewerOption3:=VIS.bGripperScrewer1Option3Show;
bGripperScrewerOption5:=VIS.bGripperScrewer1Option5Show;
bGripperScrewerOption6:=VIS.bGripperScrewer1Option6Show;
bGripperScrewerOption7:=VIS.bGripperScrewer1Option7Show;
															
bBottleDragingStationEnable:=VIS.bBottleDragingStationEnableShow;
lrBottleDragingStationVelocity:=VIS.lrBottleDragingStationVelocityShow;
															
bCapCorrectCheckEnable:=VIS.bCapCorrectCheckEnableShow;
lrCapCorrectCheckHeightPosSV:=VIS.lrCapCorrectCheckHeightPosSVShow;
bCapCorrectCheckCameraEnable:=VIS.bCapCorrectCheckCameraEnableShow;
iCapCorrectCheckCameraProgram:=VIS.iCapCorrectCheckCameraProgramShow;
															
bBottleTransferEnable:=VIS.bBottleTransferEnableShow;
nBottleTransferProgram:=VIS.nBottleTransferProgramShow;
iBottleTransferPickOffsetX:=VIS.iBottleTransferPickOffsetXShow; 		
iBottleTransferPickOffsetY:=VIS.iBottleTransferPickOffsetYShow; 		
iBottleTransferPickOffsetZ:=VIS.iBottleTransferPickOffsetZShow;		
iBottleTransferPick2OffsetX:=VIS.iBottleTransferPick2OffsetXShow;	
iBottleTransferPick2OffsetY:=VIS.iBottleTransferPick2OffsetYShow;		
iBottleTransferPick2OffsetZ:=VIS.iBottleTransferPick2OffsetZShow;		
iBottleTransferPlace1OffsetX:=VIS.iBottleTransferPlace1OffsetXShow; 	
iBottleTransferPlace1OffsetY:=VIS.iBottleTransferPlace1OffsetYShow; 	
iBottleTransferPlace1OffsetZ:=VIS.iBottleTransferPlace1OffsetZShow;	
iBottleTransferPlace2OffsetX:=VIS.iBottleTransferPlace2OffsetXShow;	
iBottleTransferPlace2OffsetY:=VIS.iBottleTransferPlace2OffsetYShow;	
iBottleTransferPlace2OffsetZ:=VIS.iBottleTransferPlace2OffsetZShow; 	
iBottleTransferSpeed:=VIS.iBottleTransferSpeedShow;			
bBottleTransferInkJetEnable:=VIS.bBottleTransferInkJetEnableShow;	
bBottleTransferPickOnlyOne:=VIS.bBottleTransferPickOnlyOneShow;		
bBottleTransferWeightEnable:=VIS.bBottleTransferWeightEnableShow;			
iBottleTransferWeightInterval:=VIS.iBottleTransferWeightIntervalShow;	
		
bBottleTransferAfterDragEnable:= VIS.bBottleTransferAfterDragEnableShow;
												
bBadBottleConveyorEnable:=VIS.bFormTransportersEnableShow:=NOT bTestTransporter;
nBadBottleConveyorVelocitySV:=VIS.nBadBottleConveyorVelocitySVShow;
															
bLabelMachineEnable:=VIS.bLabelMachineEnableShow;
															
bExitTurnTableEnable:=VIS.bExitTurnTable1EnableShow;
bExitConveyorEnable:=VIS.bExitConveyorEnableShow;
nExitConveyorVelocitySV:=VIS.nExitConveyorVelocitySVShow;	
	
														
bFormTransportersEnable:=VIS.bFormTransportersEnableShow;
nFormTransportersDispencerVelocitySV:=VIS.nFormTransportersDispencerVelocitySVShow;
//Przed ROPP
nFormTransportersROPPVelocitySV			:=	VIS.nFormTransportersROPPVelocitySVShow;
//Za ROPP
nFormTransportersScrewerVelocitySV		:=	VIS.nFormTransportersScrewerVelocitySVShow;

IF P00_PackML.tonbCapSorterOrCapSorterDragError.Q OR P00_PackML.tofFormTransportersScrewerSlowSpeed.Q 
OR P00_PackML.fbTransporterQueues.bOut // Blokada kolejek do testów
THEN
	nFormTransportersScrewerVelocitySV	:= 300; 
	nFormTransportersROPPVelocitySV		:= 300; 
END_IF	

//IF NOT P00_PackML.bDelayAfterStartFullRegister THEN	;//nFormTransportersSlowerVelocitySV	:=	600;ELSE	;//nFormTransportersSlowerVelocitySV	:=	VIS.nFormTransportersSlowerVelocitySVShow;	END_IF

nFormTransportersAfterCapSorterVelocitySV:=VIS.nFormTransportersAfterCapSorterVelocitySVShow;
nFormTransportersBeforeScrewerVelocitySV:=VIS.nFormTransportersBeforeScrewerVelocitySVShow;

nFormTransportersAfterScrewerVelocitySV:=VIS.nFormTransportersAfterScrewerVelocitySVShow;
IF bFormTransportersDispencerSlowSpeed THEN
	nFormTransportersAfterScrewerVelocitySV := 600;// bylo 600;	
END_IF
IF bDosingTwoPhases THEN
	nFormTransportersAfterScrewerVelocitySV := 550;// bylo 600;	
END_IF
														
bCircularInkjetEnable:=VIS.bCircularInkjetEnableShow;	
iCircularInkjetSpeed:=VIS.iCircularInkjetSpeedShow;
iCircularInkjetDelay:=VIS.iCircularInkjetDelayShow;	
iCircularInkjetHold:=VIS.iCircularInkjetHoldShow;
END_ACTION

ACTION aTwoSpeeds:


bFastSpeed := FALSE;//NOT VIS.bBadBottleConveyorEnableShow;

//IF NOT bFastSpeed THEN //Wolna prędkość
	
	VIS.lrFormsDragingRightVelocityShow					:=	500;
	VIS.lrFormsDragingRightAccelerationShow				:= 1200;
	VIS.lrFormsDragingRightDecelerationShow				:= 900;
	                                        			
	VIS.lrFormsDragingLeftVelocityShow					:=	500;
	VIS.lrFormsDragingLeftAccelerationShow				:= 1200;
	VIS.lrFormsDragingLeftDecelerationShow				:= 900;
	                                        			
	VIS.lrLidSealerDragingStationVelocityShow			:= 660;
	VIS.lrLidSealerDragingStationAccelerationShow		:= 2500;//1500;
	VIS.lrLidSealerDragingStationDecelerationShow  		:= 2500;//1500;
	
	VIS.lrLidFeederDragingStationVelocityShow			:= 660;
	VIS.lrLidFeederDragingStationAccelerationShow	    := 1500;
	VIS.lrLidFeederDragingStationDecelerationShow	    := 1500;
	
	VIS_ROPP.lrROPPDragVelocityShow						:=  350;
	VIS_ROPP.lrROPPDragAccelerationShow					:= 	1200;
	VIS_ROPP.lrROPPDragDecelerationShow					:= 	900;	
	VIS_ROPP.nROPPSlowerVelocitySVShow 					:=	1700;
	
	VIS.lrCapSorterDragVelocityShow						:=	500;
	VIS.lrCapSorterDragAccelerationShow					:=  1200; //bylo 1200
	VIS.lrCapSorterDragDecelerationShow					:= 	1200; //bylo 900
	                                        			
	VIS.lrBottleDragingStationVelocityShow				:=	520;	
	
	IF NOT vis.bDosingTwoPhasesShow THEN
	VIS.nFormTransportersDispencerVelocitySVShow		:= 1130; //1400	//bylo 1000
	VIS.nFormTransportersAfterScrewerVelocitySVShow		:= 850;	// bylo 1000;
	ELSE
	VIS.nFormTransportersDispencerVelocitySVShow		:= 720;
 	VIS.nFormTransportersAfterScrewerVelocitySVShow		:= 930 ;	
	END_IF 
	
	IF bChangeOver AND NOT VIS.bWeighingForm THEN
		VIS.nFormTransportersDispencerVelocitySVShow		:= 300;		
	END_IF

	IF bLidFeederEnable THEN
		VIS.nFormTransportersAfterScrewerVelocitySVShow	:= 1130;   
		VIS.nFormTransportersBeforeScrewerVelocitySVShow:= 700;     
	END_IF	
	
	//VIS.nFormTransportersScrewerVelocitySVShow		:= 620;
	//VIS.nFormTransportersBeforeScrewerVelocitySVShow	:= 600;


	VIS.nFormTransportersBeforeScrewerVelocitySVShow	:= 750 ;	//620
	VIS.nFormTransportersSlowerVelocitySVShow 			:= 2000;
	VIS.nFormTransportersROPPVelocitySVShow				:= 720;  //Przed ROPP
	VIS.nFormTransportersScrewerVelocitySVShow			:= 720;// 884 ; //Za ROPP
	VIS.nBadBottleConveyorVelocitySVShow				:= 1400;
//ELSE
//	VIS.lrFormsDragingRightVelocityShow					:=	520;//500;
//	VIS.lrFormsDragingRightAccelerationShow				:= 1200;
//	VIS.lrFormsDragingRightDecelerationShow				:= 1200;
//	                                        			
//	VIS.lrFormsDragingLeftVelocityShow					:=	520;//500;
//	VIS.lrFormsDragingLeftAccelerationShow				:= 1200;
//	VIS.lrFormsDragingLeftDecelerationShow				:= 1200;
//	                                        			
//	VIS.lrCapSorterDragVelocityShow						:=	600;//500;
//	VIS.lrCapSorterDragAccelerationShow					:= 	1200;
//	VIS.lrCapSorterDragDecelerationShow					:= 	1200;
//
//	VIS_ROPP.lrROPPDragVelocityShow						:=	500;
//	VIS_ROPP.lrROPPDragAccelerationShow					:= 	1200;
//	VIS_ROPP.lrROPPDragDecelerationShow					:= 	900;	
//	VIS_ROPP.nROPPSlowerVelocitySVShow 					:=	2100;
//	                                        			
//	VIS.lrBottleDragingStationVelocityShow				:=	500;	
//
//	VIS.nFormTransportersDispencerVelocitySVShow		:= 1300;
//	VIS.nFormTransportersScrewerVelocitySVShow			:= 900;
//	VIS.nFormTransportersBeforeScrewerVelocitySVShow	:= 830;
//	VIS.nBadBottleConveyorVelocitySVShow				:= 1200;
//	
//	//IF bFormTransportersDispencerSlowSpeed THEN
//	//	nFormTransportersDispencerVelocitySV := 1030;// bylo 600;
//	//END_IF
//END_IF
END_ACTION

END_PROGRAM

// ---- POUs/FB/Various/FB_Skalowanie.TcPOU
FUNCTION_BLOCK FB_Skalowanie
VAR_INPUT
	Ymax: REAL;
	Xmax: REAL;
	Xmin: REAL;
	Ymin: REAL;
	X: REAL;
END_VAR
VAR_OUTPUT
	Y: REAL;
	bAlarmLo: BOOL;
	bALarmHi: BOOL;
END_VAR
VAR
	A: REAL;
	B: REAL;
END_VAR

IF X<=Xmin THEN
	
	Y:=Ymin;
	bAlarmLo:=TRUE;
	bALarmHi:=FALSE;

ELSIF X>=Xmax THEN
	
	Y:=Ymax;
	bAlarmLo:=FALSE;
	bALarmHi:=TRUE;

ELSE
	IF Xmax<> Xmin THEN
	
		A:=(Ymax-Ymin)/(Xmax-Xmin);
		B:=Ymax-A*Xmax;
		Y:=A*X+B;
		bAlarmLo:=FALSE;
		bALarmHi:=FALSE;
		
	ELSE
		
		Y:=Ymax;
		bAlarmLo:=TRUE;
		bALarmHi:=TRUE;
		
	END_IF;
END_IF;

END_FUNCTION_BLOCK

// ---- POUs/P01_BottleSorter.TcPOU
PROGRAM P01_BottleSorter
VAR
END_VAR

aBottleSorterWarnings();

ACTION aBottleSorterWarnings:
//Warning 0

IF (stBottleSorterRead.eReservedSignals.iReserved20.0 AND stBottleSorterRead.bEnable) AND NOT BottleSorterWarning[0].bWarning THEN
	BottleSorterWarning[0].bWarning											:=TRUE;
	BottleSorterWarning[0].udiWarningCode									:=9;
	BottleSorterWarning[0].sDescription										:='Sorter butelek | Brak butelek w zasobniku';
ELSIF NOT stBottleSorterRead.eReservedSignals.iReserved20.0 AND BottleSorterWarning[0].bAcknowledge THEN
	BottleSorterWarning[0].bWarning											:=FALSE;
	BottleSorterWarning[0].bAcknowledge										:=FALSE;
	VIS.uliWarningAcknowledge.33											:=FALSE;
ELSIF BottleSorterWarning[0].bAcknowledge THEN                                
	BottleSorterWarning[0].bAcknowledge										:=TRUE;
END_IF

//Warning 1
IF stBottleSorterRead.eReservedSignals.iReserved20.1 AND NOT BottleSorterWarning[1].bWarning THEN
	BottleSorterWarning[1].bWarning											:=TRUE;
	BottleSorterWarning[1].udiWarningCode									:=10;
	BottleSorterWarning[1].sDescription										:='Sorter butelek | warning 1';
ELSIF NOT stBottleSorterRead.eReservedSignals.iReserved20.1 AND BottleSorterWarning[1].bAcknowledge THEN
	BottleSorterWarning[1].bWarning											:=FALSE;
	BottleSorterWarning[1].bAcknowledge										:=FALSE;
	VIS.uliWarningAcknowledge.34											:=FALSE;
ELSIF BottleSorterWarning[1].bAcknowledge THEN                                
	BottleSorterWarning[1].bAcknowledge										:=TRUE;
END_IF

//Warning 2
IF stBottleSorterRead.eReservedSignals.iReserved20.2 AND NOT BottleSorterWarning[2].bWarning THEN
	BottleSorterWarning[2].bWarning											:=TRUE;
	BottleSorterWarning[2].udiWarningCode									:=11;
	BottleSorterWarning[2].sDescription										:='Sorter butelek | warning 2';
ELSIF NOT stBottleSorterRead.eReservedSignals.iReserved20.1 AND BottleSorterWarning[2].bAcknowledge THEN
	BottleSorterWarning[2].bWarning											:=FALSE;
	BottleSorterWarning[2].bAcknowledge										:=FALSE;
	VIS.uliWarningAcknowledge.35											:=FALSE;
ELSIF BottleSorterWarning[2].bAcknowledge THEN                                
	BottleSorterWarning[2].bAcknowledge										:=TRUE;
END_IF

//Warning 3
IF stBottleSorterRead.eReservedSignals.iReserved20.3 AND NOT BottleSorterWarning[3].bWarning THEN
	BottleSorterWarning[3].bWarning											:=TRUE;
	BottleSorterWarning[3].udiWarningCode									:=12;
	BottleSorterWarning[3].sDescription										:='Sorter butelek | warning 3';
ELSIF NOT stBottleSorterRead.eReservedSignals.iReserved20.1 AND BottleSorterWarning[3].bAcknowledge THEN
	BottleSorterWarning[3].bWarning											:=FALSE;
	BottleSorterWarning[3].bAcknowledge										:=FALSE;
	VIS.uliWarningAcknowledge.36											:=FALSE;
ELSIF BottleSorterWarning[3].bAcknowledge THEN                                
	BottleSorterWarning[3].bAcknowledge										:=TRUE;
END_IF

//Warning 4
IF stBottleSorterRead.eReservedSignals.iReserved20.4 AND NOT BottleSorterWarning[4].bWarning THEN
	BottleSorterWarning[4].bWarning											:=TRUE;
	BottleSorterWarning[4].udiWarningCode									:=13;
	BottleSorterWarning[4].sDescription										:='Sorter butelek | warning 4';
ELSIF NOT stBottleSorterRead.eReservedSignals.iReserved20.1 AND BottleSorterWarning[4].bAcknowledge THEN
	BottleSorterWarning[4].bWarning											:=FALSE;
	BottleSorterWarning[4].bAcknowledge										:=FALSE;
	VIS.uliWarningAcknowledge.37											:=FALSE;
ELSIF BottleSorterWarning[4].bAcknowledge THEN
	BottleSorterWarning[4].bAcknowledge										:=TRUE;
END_IF

//Warning 5
IF stBottleSorterRead.eReservedSignals.iReserved20.5 AND NOT BottleSorterWarning[5].bWarning THEN
	BottleSorterWarning[5].bWarning											:=TRUE;
	BottleSorterWarning[5].udiWarningCode									:=14;
	BottleSorterWarning[5].sDescription										:='Sorter butelek | warning 5';
ELSIF NOT stBottleSorterRead.eReservedSignals.iReserved20.1 AND BottleSorterWarning[5].bAcknowledge THEN
	BottleSorterWarning[5].bWarning											:=FALSE;
	BottleSorterWarning[5].bAcknowledge										:=FALSE;
	VIS.uliWarningAcknowledge.38											:=FALSE;
ELSIF BottleSorterWarning[5].bAcknowledge THEN
	BottleSorterWarning[5].bAcknowledge										:=TRUE;
END_IF
END_ACTION

END_PROGRAM

// ---- POUs/P05_WeightCorrection.TcPOU
(*
Nazwa:			P05_WeightCorrection
Opis:			Stacja korekcji wagi
Wersja:			v0.1
Data:			2019-11-05
Autor:			DP
Urzadzenia:		
Konfiguracja:	
Info:
- przeróbka na RFID
- sprawdzone dwufazowe
*)
PROGRAM P05_WeightCorrection
VAR
	fbDispencer1Correction:FB_WeightCorrection;
	fbDispencer2Correction:FB_WeightCorrection;
	fbDispencer3Correction:FB_WeightCorrection;
	fbDispencer4Correction:FB_WeightCorrection;
	rtAddMeasurmen: R_TRIG;
	i: UINT;
	i2: UINT;
	i3: UINT;
	i4: UINT;
	i5: UINT;
	nCountCheck600: INT;
	rtWeightingDone: R_TRIG;

		
	k1: UINT;
	k2: UINT;
	k3: UINT;
	k4: UINT;
	nCountCheck700: INT;
	nCountCheck800: INT;
	nCountCheck900: INT;
	rtAddMeasurmen1: R_TRIG;
	rtAddMeasurmen2: R_TRIG;
	rtAddMeasurmen3: R_TRIG;
	rtAddMeasurmen4: R_TRIG;
	iCorectTest: INT;
	iCorectTest2: INT;
	iCorectTest3: INT;
	iCorectTest4: INT;
	iCorectTest5: INT;
	iCorectTest6: INT;
	iCorectTest7: INT;
	iCorectTest8: INT;
	
END_VAR

(**** Korekcja zależnie od wielkości dozy****)
IF lrDispencer1DoseVolume < 40 THEN
	
	fbDispencer1Correction.lrCorrectionStep 								:= 0.5;
	fbDispencer2Correction.lrCorrectionStep 								:= 0.5;
	fbDispencer3Correction.lrCorrectionStep 								:= 0.5;
	fbDispencer3Correction.lrCorrectionStep 								:= 0.5;
	
ELSE
	
	fbDispencer1Correction.lrCorrectionStep 								:= 1;
	fbDispencer2Correction.lrCorrectionStep 								:= 1;	
	fbDispencer3Correction.lrCorrectionStep 								:= 1;
	fbDispencer4Correction.lrCorrectionStep 								:= 1;
	
END_IF
(**** Koniec Korekcja zależnie od wielkości dozy****)


(***********Generowanie pomiarów do korekty******************)
IF bDosingTwoPhases THEN
	rtWeightingDone(CLK:=eWeightPackage2PhasePackageState[1].bWeighed,Q=>); //Triger dodania wagi do korekty
	TwoPhaseDosing();
ELSE
	rtWeightingDone(CLK:=eWeightPackageState[1].bWeighed,Q=>); //Triger dodania wagi do korekty
	OnePhaseDosing();
END_IF
(***********Koniec Generowanie pomiarów do korekty******************)
	

// Wpisywanie odpowiednich wag zadanych do bloku korekci
IF VIS.bDosingTwoPhasesShow THEN
	
	fbDispencer1Correction.lrActualDoseVolumeSV 					:= lrDispencer1DoseVolume + lrDispencer2DoseVolume + VIS.lrDispencer1CorrectionWeight;
	fbDispencer2Correction.lrActualDoseVolumeSV 					:= lrDispencer1DoseVolume + lrDispencer2DoseVolume + VIS.lrDispencer2CorrectionWeight;
	fbDispencer3Correction.lrActualDoseVolumeSV 					:= lrDispencer1DoseVolume + lrDispencer2DoseVolume + VIS.lrDispencer3CorrectionWeight;
	fbDispencer4Correction.lrActualDoseVolumeSV 					:= lrDispencer1DoseVolume + lrDispencer2DoseVolume + VIS.lrDispencer4CorrectionWeight;		
ELSE
	fbDispencer1Correction.lrActualDoseVolumeSV 					:= lrDispencer1DoseVolume + VIS.lrDispencer1CorrectionWeight;
	fbDispencer2Correction.lrActualDoseVolumeSV 					:= lrDispencer1DoseVolume + VIS.lrDispencer2CorrectionWeight;
	fbDispencer3Correction.lrActualDoseVolumeSV 					:= lrDispencer1DoseVolume + VIS.lrDispencer3CorrectionWeight;
	fbDispencer4Correction.lrActualDoseVolumeSV 					:= lrDispencer1DoseVolume + VIS.lrDispencer4CorrectionWeight;		
END_IF
(**Zabezpieczenie przed błędną wartością w tablicy***)
IF k1=0 THEN	k1:=1;END_IF
IF k2=0 THEN	k2:=1;END_IF
IF k3=0 THEN	k3:=1;END_IF
IF k4=0 THEN	k4:=1;END_IF

(******bloki korekcji****)												
Correction();
VIS.bWeightCorrectionReset:=FALSE; 

//Diagnostyka
rtAddMeasurmen1(CLK:=fbDispencer1Correction.bAddMeasurment,Q=>);
IF rtAddMeasurmen1.Q THEN
	nCountCheck600												:= nCountCheck600+1;
END_IF

rtAddMeasurmen2(CLK:=fbDispencer2Correction.bAddMeasurment,Q=>);
IF rtAddMeasurmen2.Q THEN
	nCountCheck700												:= nCountCheck700+1;
END_IF

rtAddMeasurmen3(CLK:=fbDispencer3Correction.bAddMeasurment,Q=>);
IF rtAddMeasurmen3.Q THEN
	nCountCheck800												:= nCountCheck800+1;
END_IF

rtAddMeasurmen4(CLK:=fbDispencer4Correction.bAddMeasurment,Q=>);
IF rtAddMeasurmen4.Q THEN
	nCountCheck900												:= nCountCheck900+1;
END_IF
	
(**Kasowanie wartości przy dozowaniu dwufazowym***)
fbDispencer1Correction.bAddMeasurment 							:= FALSE;
fbDispencer2Correction.bAddMeasurment 							:= FALSE;
fbDispencer3Correction.bAddMeasurment 							:= FALSE;
fbDispencer4Correction.bAddMeasurment 							:= FALSE;

